	{attribute	'TcLinkTo'	:=	'.Status:=TIIB[LAMP_CLSTR1_PNL1_EP03_EP6002-0002]^COM TxPDO-Map Inputs Channel 1^Status;
								 .D[0]:=TIIB[LAMP_CLSTR1_PNL1_EP03_EP6002-0002]^COM TxPDO-Map Inputs Channel 1^Data In 0;
								 .D[1]:=TIIB[LAMP_CLSTR1_PNL1_EP03_EP6002-0002]^COM TxPDO-Map Inputs Channel 1^Data In 1;
								 .D[2]:=TIIB[LAMP_CLSTR1_PNL1_EP03_EP6002-0002]^COM TxPDO-Map Inputs Channel 1^Data In 2;
								 .D[3]:=TIIB[LAMP_CLSTR1_PNL1_EP03_EP6002-0002]^COM TxPDO-Map Inputs Channel 1^Data In 3;
								 .D[4]:=TIIB[LAMP_CLSTR1_PNL1_EP03_EP6002-0002]^COM TxPDO-Map Inputs Channel 1^Data In 4;
								 .D[5]:=TIIB[LAMP_CLSTR1_PNL1_EP03_EP6002-0002]^COM TxPDO-Map Inputs Channel 1^Data In 5;
								 .D[6]:=TIIB[LAMP_CLSTR1_PNL1_EP03_EP6002-0002]^COM TxPDO-Map Inputs Channel 1^Data In 6;
								 .D[7]:=TIIB[LAMP_CLSTR1_PNL1_EP03_EP6002-0002]^COM TxPDO-Map Inputs Channel 1^Data In 7;
								 .D[8]:=TIIB[LAMP_CLSTR1_PNL1_EP03_EP6002-0002]^COM TxPDO-Map Inputs Channel 1^Data In 8;
								 .D[9]:=TIIB[LAMP_CLSTR1_PNL1_EP03_EP6002-0002]^COM TxPDO-Map Inputs Channel 1^Data In 9;
								 .D[10]:=TIIB[LAMP_CLSTR1_PNL1_EP03_EP6002-0002]^COM TxPDO-Map Inputs Channel 1^Data In 10;
								 .D[11]:=TIIB[LAMP_CLSTR1_PNL1_EP03_EP6002-0002]^COM TxPDO-Map Inputs Channel 1^Data In 11;
								 .D[12]:=TIIB[LAMP_CLSTR1_PNL1_EP03_EP6002-0002]^COM TxPDO-Map Inputs Channel 1^Data In 12;
								 .D[13]:=TIIB[LAMP_CLSTR1_PNL1_EP03_EP6002-0002]^COM TxPDO-Map Inputs Channel 1^Data In 13;
								 .D[14]:=TIIB[LAMP_CLSTR1_PNL1_EP03_EP6002-0002]^COM TxPDO-Map Inputs Channel 1^Data In 14;
								 .D[15]:=TIIB[LAMP_CLSTR1_PNL1_EP03_EP6002-0002]^COM TxPDO-Map Inputs Channel 1^Data In 15;
								 .D[16]:=TIIB[LAMP_CLSTR1_PNL1_EP03_EP6002-0002]^COM TxPDO-Map Inputs Channel 1^Data In 16;
								 .D[17]:=TIIB[LAMP_CLSTR1_PNL1_EP03_EP6002-0002]^COM TxPDO-Map Inputs Channel 1^Data In 17;
								 .D[18]:=TIIB[LAMP_CLSTR1_PNL1_EP03_EP6002-0002]^COM TxPDO-Map Inputs Channel 1^Data In 18;
								 .D[19]:=TIIB[LAMP_CLSTR1_PNL1_EP03_EP6002-0002]^COM TxPDO-Map Inputs Channel 1^Data In 19;
								 .D[20]:=TIIB[LAMP_CLSTR1_PNL1_EP03_EP6002-0002]^COM TxPDO-Map Inputs Channel 1^Data In 20;
								 .D[21]:=TIIB[LAMP_CLSTR1_PNL1_EP03_EP6002-0002]^COM TxPDO-Map Inputs Channel 1^Data In 21
	'}
	stComIn_LAMP_CLSTR1_PTM_01		AT %I*	:	EL6inData22B;
	
	{attribute	'TcLinkTo'	:=	'.Ctrl:=TIIB[LAMP_CLSTR1_PNL1_EP03_EP6002-0002]^COM RxPDO-Map Outputs Channel 1^Ctrl;
								 .D[0]:=TIIB[LAMP_CLSTR1_PNL1_EP03_EP6002-0002]^COM RxPDO-Map Outputs Channel 1^Data Out 0;
								 .D[1]:=TIIB[LAMP_CLSTR1_PNL1_EP03_EP6002-0002]^COM RxPDO-Map Outputs Channel 1^Data Out 1;
								 .D[2]:=TIIB[LAMP_CLSTR1_PNL1_EP03_EP6002-0002]^COM RxPDO-Map Outputs Channel 1^Data Out 2;
								 .D[3]:=TIIB[LAMP_CLSTR1_PNL1_EP03_EP6002-0002]^COM RxPDO-Map Outputs Channel 1^Data Out 3;
								 .D[4]:=TIIB[LAMP_CLSTR1_PNL1_EP03_EP6002-0002]^COM RxPDO-Map Outputs Channel 1^Data Out 4;
								 .D[5]:=TIIB[LAMP_CLSTR1_PNL1_EP03_EP6002-0002]^COM RxPDO-Map Outputs Channel 1^Data Out 5;
								 .D[6]:=TIIB[LAMP_CLSTR1_PNL1_EP03_EP6002-0002]^COM RxPDO-Map Outputs Channel 1^Data Out 6;
								 .D[7]:=TIIB[LAMP_CLSTR1_PNL1_EP03_EP6002-0002]^COM RxPDO-Map Outputs Channel 1^Data Out 7;
								 .D[8]:=TIIB[LAMP_CLSTR1_PNL1_EP03_EP6002-0002]^COM RxPDO-Map Outputs Channel 1^Data Out 8;
								 .D[9]:=TIIB[LAMP_CLSTR1_PNL1_EP03_EP6002-0002]^COM RxPDO-Map Outputs Channel 1^Data Out 9;
								 .D[10]:=TIIB[LAMP_CLSTR1_PNL1_EP03_EP6002-0002]^COM RxPDO-Map Outputs Channel 1^Data Out 10;
								 .D[11]:=TIIB[LAMP_CLSTR1_PNL1_EP03_EP6002-0002]^COM RxPDO-Map Outputs Channel 1^Data Out 11;
								 .D[12]:=TIIB[LAMP_CLSTR1_PNL1_EP03_EP6002-0002]^COM RxPDO-Map Outputs Channel 1^Data Out 12;
								 .D[13]:=TIIB[LAMP_CLSTR1_PNL1_EP03_EP6002-0002]^COM RxPDO-Map Outputs Channel 1^Data Out 13;
								 .D[14]:=TIIB[LAMP_CLSTR1_PNL1_EP03_EP6002-0002]^COM RxPDO-Map Outputs Channel 1^Data Out 14;
								 .D[15]:=TIIB[LAMP_CLSTR1_PNL1_EP03_EP6002-0002]^COM RxPDO-Map Outputs Channel 1^Data Out 15;
								 .D[16]:=TIIB[LAMP_CLSTR1_PNL1_EP03_EP6002-0002]^COM RxPDO-Map Outputs Channel 1^Data Out 16;
								 .D[17]:=TIIB[LAMP_CLSTR1_PNL1_EP03_EP6002-0002]^COM RxPDO-Map Outputs Channel 1^Data Out 17;
								 .D[18]:=TIIB[LAMP_CLSTR1_PNL1_EP03_EP6002-0002]^COM RxPDO-Map Outputs Channel 1^Data Out 18;
								 .D[19]:=TIIB[LAMP_CLSTR1_PNL1_EP03_EP6002-0002]^COM RxPDO-Map Outputs Channel 1^Data Out 19;
								 .D[20]:=TIIB[LAMP_CLSTR1_PNL1_EP03_EP6002-0002]^COM RxPDO-Map Outputs Channel 1^Data Out 20;
								 .D[21]:=TIIB[LAMP_CLSTR1_PNL1_EP03_EP6002-0002]^COM RxPDO-Map Outputs Channel 1^Data Out 21
	'}
	stComOut_LAMP_CLSTR1_PTM_01		AT %Q*	:	EL6outData22B;
	
	{attribute	'TcLinkTo'	:=	'.Status:=TIIB[LAMP_CLSTR1_PNL2_EP03_EP6002-0002]^COM TxPDO-Map Inputs Channel 1^Status;
								 .D[0]:=TIIB[LAMP_CLSTR1_PNL2_EP03_EP6002-0002]^COM TxPDO-Map Inputs Channel 1^Data In 0;
								 .D[1]:=TIIB[LAMP_CLSTR1_PNL2_EP03_EP6002-0002]^COM TxPDO-Map Inputs Channel 1^Data In 1;
								 .D[2]:=TIIB[LAMP_CLSTR1_PNL2_EP03_EP6002-0002]^COM TxPDO-Map Inputs Channel 1^Data In 2;
								 .D[3]:=TIIB[LAMP_CLSTR1_PNL2_EP03_EP6002-0002]^COM TxPDO-Map Inputs Channel 1^Data In 3;
								 .D[4]:=TIIB[LAMP_CLSTR1_PNL2_EP03_EP6002-0002]^COM TxPDO-Map Inputs Channel 1^Data In 4;
								 .D[5]:=TIIB[LAMP_CLSTR1_PNL2_EP03_EP6002-0002]^COM TxPDO-Map Inputs Channel 1^Data In 5;
								 .D[6]:=TIIB[LAMP_CLSTR1_PNL2_EP03_EP6002-0002]^COM TxPDO-Map Inputs Channel 1^Data In 6;
								 .D[7]:=TIIB[LAMP_CLSTR1_PNL2_EP03_EP6002-0002]^COM TxPDO-Map Inputs Channel 1^Data In 7;
								 .D[8]:=TIIB[LAMP_CLSTR1_PNL2_EP03_EP6002-0002]^COM TxPDO-Map Inputs Channel 1^Data In 8;
								 .D[9]:=TIIB[LAMP_CLSTR1_PNL2_EP03_EP6002-0002]^COM TxPDO-Map Inputs Channel 1^Data In 9;
								 .D[10]:=TIIB[LAMP_CLSTR1_PNL2_EP03_EP6002-0002]^COM TxPDO-Map Inputs Channel 1^Data In 10;
								 .D[11]:=TIIB[LAMP_CLSTR1_PNL2_EP03_EP6002-0002]^COM TxPDO-Map Inputs Channel 1^Data In 11;
								 .D[12]:=TIIB[LAMP_CLSTR1_PNL2_EP03_EP6002-0002]^COM TxPDO-Map Inputs Channel 1^Data In 12;
								 .D[13]:=TIIB[LAMP_CLSTR1_PNL2_EP03_EP6002-0002]^COM TxPDO-Map Inputs Channel 1^Data In 13;
								 .D[14]:=TIIB[LAMP_CLSTR1_PNL2_EP03_EP6002-0002]^COM TxPDO-Map Inputs Channel 1^Data In 14;
								 .D[15]:=TIIB[LAMP_CLSTR1_PNL2_EP03_EP6002-0002]^COM TxPDO-Map Inputs Channel 1^Data In 15;
								 .D[16]:=TIIB[LAMP_CLSTR1_PNL2_EP03_EP6002-0002]^COM TxPDO-Map Inputs Channel 1^Data In 16;
								 .D[17]:=TIIB[LAMP_CLSTR1_PNL2_EP03_EP6002-0002]^COM TxPDO-Map Inputs Channel 1^Data In 17;
								 .D[18]:=TIIB[LAMP_CLSTR1_PNL2_EP03_EP6002-0002]^COM TxPDO-Map Inputs Channel 1^Data In 18;
								 .D[19]:=TIIB[LAMP_CLSTR1_PNL2_EP03_EP6002-0002]^COM TxPDO-Map Inputs Channel 1^Data In 19;
								 .D[20]:=TIIB[LAMP_CLSTR1_PNL2_EP03_EP6002-0002]^COM TxPDO-Map Inputs Channel 1^Data In 20;
								 .D[21]:=TIIB[LAMP_CLSTR1_PNL2_EP03_EP6002-0002]^COM TxPDO-Map Inputs Channel 1^Data In 21
	'}
	stComIn_LAMP_CLSTR1_PTM_02		AT %I*	:	EL6inData22B;
	
	{attribute	'TcLinkTo'	:=	'.Ctrl:=TIIB[LAMP_CLSTR1_PNL2_EP03_EP6002-0002]^COM RxPDO-Map Outputs Channel 1^Ctrl;
								 .D[0]:=TIIB[LAMP_CLSTR1_PNL2_EP03_EP6002-0002]^COM RxPDO-Map Outputs Channel 1^Data Out 0;
								 .D[1]:=TIIB[LAMP_CLSTR1_PNL2_EP03_EP6002-0002]^COM RxPDO-Map Outputs Channel 1^Data Out 1;
								 .D[2]:=TIIB[LAMP_CLSTR1_PNL2_EP03_EP6002-0002]^COM RxPDO-Map Outputs Channel 1^Data Out 2;
								 .D[3]:=TIIB[LAMP_CLSTR1_PNL2_EP03_EP6002-0002]^COM RxPDO-Map Outputs Channel 1^Data Out 3;
								 .D[4]:=TIIB[LAMP_CLSTR1_PNL2_EP03_EP6002-0002]^COM RxPDO-Map Outputs Channel 1^Data Out 4;
								 .D[5]:=TIIB[LAMP_CLSTR1_PNL2_EP03_EP6002-0002]^COM RxPDO-Map Outputs Channel 1^Data Out 5;
								 .D[6]:=TIIB[LAMP_CLSTR1_PNL2_EP03_EP6002-0002]^COM RxPDO-Map Outputs Channel 1^Data Out 6;
								 .D[7]:=TIIB[LAMP_CLSTR1_PNL2_EP03_EP6002-0002]^COM RxPDO-Map Outputs Channel 1^Data Out 7;
								 .D[8]:=TIIB[LAMP_CLSTR1_PNL2_EP03_EP6002-0002]^COM RxPDO-Map Outputs Channel 1^Data Out 8;
								 .D[9]:=TIIB[LAMP_CLSTR1_PNL2_EP03_EP6002-0002]^COM RxPDO-Map Outputs Channel 1^Data Out 9;
								 .D[10]:=TIIB[LAMP_CLSTR1_PNL2_EP03_EP6002-0002]^COM RxPDO-Map Outputs Channel 1^Data Out 10;
								 .D[11]:=TIIB[LAMP_CLSTR1_PNL2_EP03_EP6002-0002]^COM RxPDO-Map Outputs Channel 1^Data Out 11;
								 .D[12]:=TIIB[LAMP_CLSTR1_PNL2_EP03_EP6002-0002]^COM RxPDO-Map Outputs Channel 1^Data Out 12;
								 .D[13]:=TIIB[LAMP_CLSTR1_PNL2_EP03_EP6002-0002]^COM RxPDO-Map Outputs Channel 1^Data Out 13;
								 .D[14]:=TIIB[LAMP_CLSTR1_PNL2_EP03_EP6002-0002]^COM RxPDO-Map Outputs Channel 1^Data Out 14;
								 .D[15]:=TIIB[LAMP_CLSTR1_PNL2_EP03_EP6002-0002]^COM RxPDO-Map Outputs Channel 1^Data Out 15;
								 .D[16]:=TIIB[LAMP_CLSTR1_PNL2_EP03_EP6002-0002]^COM RxPDO-Map Outputs Channel 1^Data Out 16;
								 .D[17]:=TIIB[LAMP_CLSTR1_PNL2_EP03_EP6002-0002]^COM RxPDO-Map Outputs Channel 1^Data Out 17;
								 .D[18]:=TIIB[LAMP_CLSTR1_PNL2_EP03_EP6002-0002]^COM RxPDO-Map Outputs Channel 1^Data Out 18;
								 .D[19]:=TIIB[LAMP_CLSTR1_PNL2_EP03_EP6002-0002]^COM RxPDO-Map Outputs Channel 1^Data Out 19;
								 .D[20]:=TIIB[LAMP_CLSTR1_PNL2_EP03_EP6002-0002]^COM RxPDO-Map Outputs Channel 1^Data Out 20;
								 .D[21]:=TIIB[LAMP_CLSTR1_PNL2_EP03_EP6002-0002]^COM RxPDO-Map Outputs Channel 1^Data Out 21
	'}
	stComOut_LAMP_CLSTR1_PTM_02		AT %Q*	:	EL6outData22B;
	
	{attribute	'TcLinkTo'	:=	'.Status:=TIIB[LAMP_CLSTR1_PNL3_EP03_EP6002-0002]^COM TxPDO-Map Inputs Channel 1^Status;
								 .D[0]:=TIIB[LAMP_CLSTR1_PNL3_EP03_EP6002-0002]^COM TxPDO-Map Inputs Channel 1^Data In 0;
								 .D[1]:=TIIB[LAMP_CLSTR1_PNL3_EP03_EP6002-0002]^COM TxPDO-Map Inputs Channel 1^Data In 1;
								 .D[2]:=TIIB[LAMP_CLSTR1_PNL3_EP03_EP6002-0002]^COM TxPDO-Map Inputs Channel 1^Data In 2;
								 .D[3]:=TIIB[LAMP_CLSTR1_PNL3_EP03_EP6002-0002]^COM TxPDO-Map Inputs Channel 1^Data In 3;
								 .D[4]:=TIIB[LAMP_CLSTR1_PNL3_EP03_EP6002-0002]^COM TxPDO-Map Inputs Channel 1^Data In 4;
								 .D[5]:=TIIB[LAMP_CLSTR1_PNL3_EP03_EP6002-0002]^COM TxPDO-Map Inputs Channel 1^Data In 5;
								 .D[6]:=TIIB[LAMP_CLSTR1_PNL3_EP03_EP6002-0002]^COM TxPDO-Map Inputs Channel 1^Data In 6;
								 .D[7]:=TIIB[LAMP_CLSTR1_PNL3_EP03_EP6002-0002]^COM TxPDO-Map Inputs Channel 1^Data In 7;
								 .D[8]:=TIIB[LAMP_CLSTR1_PNL3_EP03_EP6002-0002]^COM TxPDO-Map Inputs Channel 1^Data In 8;
								 .D[9]:=TIIB[LAMP_CLSTR1_PNL3_EP03_EP6002-0002]^COM TxPDO-Map Inputs Channel 1^Data In 9;
								 .D[10]:=TIIB[LAMP_CLSTR1_PNL3_EP03_EP6002-0002]^COM TxPDO-Map Inputs Channel 1^Data In 10;
								 .D[11]:=TIIB[LAMP_CLSTR1_PNL3_EP03_EP6002-0002]^COM TxPDO-Map Inputs Channel 1^Data In 11;
								 .D[12]:=TIIB[LAMP_CLSTR1_PNL3_EP03_EP6002-0002]^COM TxPDO-Map Inputs Channel 1^Data In 12;
								 .D[13]:=TIIB[LAMP_CLSTR1_PNL3_EP03_EP6002-0002]^COM TxPDO-Map Inputs Channel 1^Data In 13;
								 .D[14]:=TIIB[LAMP_CLSTR1_PNL3_EP03_EP6002-0002]^COM TxPDO-Map Inputs Channel 1^Data In 14;
								 .D[15]:=TIIB[LAMP_CLSTR1_PNL3_EP03_EP6002-0002]^COM TxPDO-Map Inputs Channel 1^Data In 15;
								 .D[16]:=TIIB[LAMP_CLSTR1_PNL3_EP03_EP6002-0002]^COM TxPDO-Map Inputs Channel 1^Data In 16;
								 .D[17]:=TIIB[LAMP_CLSTR1_PNL3_EP03_EP6002-0002]^COM TxPDO-Map Inputs Channel 1^Data In 17;
								 .D[18]:=TIIB[LAMP_CLSTR1_PNL3_EP03_EP6002-0002]^COM TxPDO-Map Inputs Channel 1^Data In 18;
								 .D[19]:=TIIB[LAMP_CLSTR1_PNL3_EP03_EP6002-0002]^COM TxPDO-Map Inputs Channel 1^Data In 19;
								 .D[20]:=TIIB[LAMP_CLSTR1_PNL3_EP03_EP6002-0002]^COM TxPDO-Map Inputs Channel 1^Data In 20;
								 .D[21]:=TIIB[LAMP_CLSTR1_PNL3_EP03_EP6002-0002]^COM TxPDO-Map Inputs Channel 1^Data In 21
	'}
	stComIn_LAMP_CLSTR1_PTM_03		AT %I*	:	EL6inData22B;
	
	{attribute	'TcLinkTo'	:=	'.Ctrl:=TIIB[LAMP_CLSTR1_PNL3_EP03_EP6002-0002]^COM RxPDO-Map Outputs Channel 1^Ctrl;
								 .D[0]:=TIIB[LAMP_CLSTR1_PNL3_EP03_EP6002-0002]^COM RxPDO-Map Outputs Channel 1^Data Out 0;
								 .D[1]:=TIIB[LAMP_CLSTR1_PNL3_EP03_EP6002-0002]^COM RxPDO-Map Outputs Channel 1^Data Out 1;
								 .D[2]:=TIIB[LAMP_CLSTR1_PNL3_EP03_EP6002-0002]^COM RxPDO-Map Outputs Channel 1^Data Out 2;
								 .D[3]:=TIIB[LAMP_CLSTR1_PNL3_EP03_EP6002-0002]^COM RxPDO-Map Outputs Channel 1^Data Out 3;
								 .D[4]:=TIIB[LAMP_CLSTR1_PNL3_EP03_EP6002-0002]^COM RxPDO-Map Outputs Channel 1^Data Out 4;
								 .D[5]:=TIIB[LAMP_CLSTR1_PNL3_EP03_EP6002-0002]^COM RxPDO-Map Outputs Channel 1^Data Out 5;
								 .D[6]:=TIIB[LAMP_CLSTR1_PNL3_EP03_EP6002-0002]^COM RxPDO-Map Outputs Channel 1^Data Out 6;
								 .D[7]:=TIIB[LAMP_CLSTR1_PNL3_EP03_EP6002-0002]^COM RxPDO-Map Outputs Channel 1^Data Out 7;
								 .D[8]:=TIIB[LAMP_CLSTR1_PNL3_EP03_EP6002-0002]^COM RxPDO-Map Outputs Channel 1^Data Out 8;
								 .D[9]:=TIIB[LAMP_CLSTR1_PNL3_EP03_EP6002-0002]^COM RxPDO-Map Outputs Channel 1^Data Out 9;
								 .D[10]:=TIIB[LAMP_CLSTR1_PNL3_EP03_EP6002-0002]^COM RxPDO-Map Outputs Channel 1^Data Out 10;
								 .D[11]:=TIIB[LAMP_CLSTR1_PNL3_EP03_EP6002-0002]^COM RxPDO-Map Outputs Channel 1^Data Out 11;
								 .D[12]:=TIIB[LAMP_CLSTR1_PNL3_EP03_EP6002-0002]^COM RxPDO-Map Outputs Channel 1^Data Out 12;
								 .D[13]:=TIIB[LAMP_CLSTR1_PNL3_EP03_EP6002-0002]^COM RxPDO-Map Outputs Channel 1^Data Out 13;
								 .D[14]:=TIIB[LAMP_CLSTR1_PNL3_EP03_EP6002-0002]^COM RxPDO-Map Outputs Channel 1^Data Out 14;
								 .D[15]:=TIIB[LAMP_CLSTR1_PNL3_EP03_EP6002-0002]^COM RxPDO-Map Outputs Channel 1^Data Out 15;
								 .D[16]:=TIIB[LAMP_CLSTR1_PNL3_EP03_EP6002-0002]^COM RxPDO-Map Outputs Channel 1^Data Out 16;
								 .D[17]:=TIIB[LAMP_CLSTR1_PNL3_EP03_EP6002-0002]^COM RxPDO-Map Outputs Channel 1^Data Out 17;
								 .D[18]:=TIIB[LAMP_CLSTR1_PNL3_EP03_EP6002-0002]^COM RxPDO-Map Outputs Channel 1^Data Out 18;
								 .D[19]:=TIIB[LAMP_CLSTR1_PNL3_EP03_EP6002-0002]^COM RxPDO-Map Outputs Channel 1^Data Out 19;
								 .D[20]:=TIIB[LAMP_CLSTR1_PNL3_EP03_EP6002-0002]^COM RxPDO-Map Outputs Channel 1^Data Out 20;
								 .D[21]:=TIIB[LAMP_CLSTR1_PNL3_EP03_EP6002-0002]^COM RxPDO-Map Outputs Channel 1^Data Out 21
	'}
	stComOut_LAMP_CLSTR1_PTM_03		AT %Q*	:	EL6outData22B;
(*
	{attribute	'TcLinkTo'	:=	'.Status:=TIIB[KTOF_PNL1_EP03_EP6002-0002]^COM TxPDO-Map Inputs Channel 1^Status;
								 .D[0]:=TIIB[KTOF_PNL1_EP03_EP6002-0002]^COM TxPDO-Map Inputs Channel 1^Data In 0;
								 .D[1]:=TIIB[KTOF_PNL1_EP03_EP6002-0002]^COM TxPDO-Map Inputs Channel 1^Data In 1;
								 .D[2]:=TIIB[KTOF_PNL1_EP03_EP6002-0002]^COM TxPDO-Map Inputs Channel 1^Data In 2;
								 .D[3]:=TIIB[KTOF_PNL1_EP03_EP6002-0002]^COM TxPDO-Map Inputs Channel 1^Data In 3;
								 .D[4]:=TIIB[KTOF_PNL1_EP03_EP6002-0002]^COM TxPDO-Map Inputs Channel 1^Data In 4;
								 .D[5]:=TIIB[KTOF_PNL1_EP03_EP6002-0002]^COM TxPDO-Map Inputs Channel 1^Data In 5;
								 .D[6]:=TIIB[KTOF_PNL1_EP03_EP6002-0002]^COM TxPDO-Map Inputs Channel 1^Data In 6;
								 .D[7]:=TIIB[KTOF_PNL1_EP03_EP6002-0002]^COM TxPDO-Map Inputs Channel 1^Data In 7;
								 .D[8]:=TIIB[KTOF_PNL1_EP03_EP6002-0002]^COM TxPDO-Map Inputs Channel 1^Data In 8;
								 .D[9]:=TIIB[KTOF_PNL1_EP03_EP6002-0002]^COM TxPDO-Map Inputs Channel 1^Data In 9;
								 .D[10]:=TIIB[KTOF_PNL1_EP03_EP6002-0002]^COM TxPDO-Map Inputs Channel 1^Data In 10;
								 .D[11]:=TIIB[KTOF_PNL1_EP03_EP6002-0002]^COM TxPDO-Map Inputs Channel 1^Data In 11;
								 .D[12]:=TIIB[KTOF_PNL1_EP03_EP6002-0002]^COM TxPDO-Map Inputs Channel 1^Data In 12;
								 .D[13]:=TIIB[KTOF_PNL1_EP03_EP6002-0002]^COM TxPDO-Map Inputs Channel 1^Data In 13;
								 .D[14]:=TIIB[KTOF_PNL1_EP03_EP6002-0002]^COM TxPDO-Map Inputs Channel 1^Data In 14;
								 .D[15]:=TIIB[KTOF_PNL1_EP03_EP6002-0002]^COM TxPDO-Map Inputs Channel 1^Data In 15;
								 .D[16]:=TIIB[KTOF_PNL1_EP03_EP6002-0002]^COM TxPDO-Map Inputs Channel 1^Data In 16;
								 .D[17]:=TIIB[KTOF_PNL1_EP03_EP6002-0002]^COM TxPDO-Map Inputs Channel 1^Data In 17;
								 .D[18]:=TIIB[KTOF_PNL1_EP03_EP6002-0002]^COM TxPDO-Map Inputs Channel 1^Data In 18;
								 .D[19]:=TIIB[KTOF_PNL1_EP03_EP6002-0002]^COM TxPDO-Map Inputs Channel 1^Data In 19;
								 .D[20]:=TIIB[KTOF_PNL1_EP03_EP6002-0002]^COM TxPDO-Map Inputs Channel 1^Data In 20;
								 .D[21]:=TIIB[KTOF_PNL1_EP03_EP6002-0002]^COM TxPDO-Map Inputs Channel 1^Data In 21;
	'}
	stComIn_KTOF_PTM_01		AT %I*	:	EL6inData22B;

	{attribute	'TcLinkTo'	:=	'.Ctrl:=TIIB[KTOF_PNL1_EP03_EP6002-0002]^COM RxPDO-Map Outputs Channel 1^Ctrl;
								 .D[0]:=TIIB[KTOF_PNL1_EP03_EP6002-0002]^COM RxPDO-Map Outputs Channel 1^Data Out 0;
								 .D[1]:=TIIB[KTOF_PNL1_EP03_EP6002-0002]^COM RxPDO-Map Outputs Channel 1^Data Out 1;
								 .D[2]:=TIIB[KTOF_PNL1_EP03_EP6002-0002]^COM RxPDO-Map Outputs Channel 1^Data Out 2;
								 .D[3]:=TIIB[KTOF_PNL1_EP03_EP6002-0002]^COM RxPDO-Map Outputs Channel 1^Data Out 3;
								 .D[4]:=TIIB[KTOF_PNL1_EP03_EP6002-0002]^COM RxPDO-Map Outputs Channel 1^Data Out 4;
								 .D[5]:=TIIB[KTOF_PNL1_EP03_EP6002-0002]^COM RxPDO-Map Outputs Channel 1^Data Out 5;
								 .D[6]:=TIIB[KTOF_PNL1_EP03_EP6002-0002]^COM RxPDO-Map Outputs Channel 1^Data Out 6;
								 .D[7]:=TIIB[KTOF_PNL1_EP03_EP6002-0002]^COM RxPDO-Map Outputs Channel 1^Data Out 7;
								 .D[8]:=TIIB[KTOF_PNL1_EP03_EP6002-0002]^COM RxPDO-Map Outputs Channel 1^Data Out 8;
								 .D[9]:=TIIB[KTOF_PNL1_EP03_EP6002-0002]^COM RxPDO-Map Outputs Channel 1^Data Out 9;
								 .D[10]:=TIIB[KTOF_PNL1_EP03_EP6002-0002]^COM RxPDO-Map Outputs Channel 1^Data Out 10;
								 .D[11]:=TIIB[KTOF_PNL1_EP03_EP6002-0002]^COM RxPDO-Map Outputs Channel 1^Data Out 11;
								 .D[12]:=TIIB[KTOF_PNL1_EP03_EP6002-0002]^COM RxPDO-Map Outputs Channel 1^Data Out 12;
								 .D[13]:=TIIB[KTOF_PNL1_EP03_EP6002-0002]^COM RxPDO-Map Outputs Channel 1^Data Out 13;
								 .D[14]:=TIIB[KTOF_PNL1_EP03_EP6002-0002]^COM RxPDO-Map Outputs Channel 1^Data Out 14;
								 .D[15]:=TIIB[KTOF_PNL1_EP03_EP6002-0002]^COM RxPDO-Map Outputs Channel 1^Data Out 15;
								 .D[16]:=TIIB[KTOF_PNL1_EP03_EP6002-0002]^COM RxPDO-Map Outputs Channel 1^Data Out 16;
								 .D[17]:=TIIB[KTOF_PNL1_EP03_EP6002-0002]^COM RxPDO-Map Outputs Channel 1^Data Out 17;
								 .D[18]:=TIIB[KTOF_PNL1_EP03_EP6002-0002]^COM RxPDO-Map Outputs Channel 1^Data Out 18;
								 .D[19]:=TIIB[KTOF_PNL1_EP03_EP6002-0002]^COM RxPDO-Map Outputs Channel 1^Data Out 19;
								 .D[20]:=TIIB[KTOF_PNL1_EP03_EP6002-0002]^COM RxPDO-Map Outputs Channel 1^Data Out 20;
								 .D[21]:=TIIB[KTOF_PNL1_EP03_EP6002-0002]^COM RxPDO-Map Outputs Channel 1^Data Out 21;
	'}
	stComOut_KTOF_PTM_01		AT %Q*	:	EL6outData22B;
*)
	//Leybolds
	// GJ2 not included in LV17 configuration
END_VAR

// ---- GVLs/GVL_Devices.TcGVL
//{attribute 'qualified_only'}
VAR_GLOBAL
	
(*Rack Mounted Turbo Pumps*)
// GJ2 not included in LV17 configuration

(*Onboard Turbo Pumps*)
	{attribute 'TcLinkTo' := 	'.i_xAtSpd			:=	TIIB[LAMP_PNL1_EP01_EP2338-0002]^Channel 1^Input;
								 .i_xFaultNC		:=	TIIB[LAMP_PNL1_EP01_EP2338-0002]^Channel 2^Input;
								 .i_xRemote			:=	TIIB[LAMP_PNL1_EP01_EP2338-0002]^Channel 3^Input;
								 .q_RunDO			:=	TIIB[LAMP_PNL1_EP02_EP2624-0002]^Channel 1^Output;
								 .q_xReset 			:=	TIIB[LAMP_PNL1_EP02_EP2624-0002]^Channel 2^Output				 
	'}
	{attribute 'pytmc' := '
		pv: LAMP:C2:PTM:01
		io: io
	'}
	LAMP_C2_PTM_01 : FB_PTM_Pfeiffer;
	
	{attribute 'TcLinkTo' := 	'.i_xAtSpd			:=	TIIB[LAMP_PNL1_EP01_EP2338-0002]^Channel 5^Input;
								 .i_xFaultNC		:=	TIIB[LAMP_PNL1_EP01_EP2338-0002]^Channel 6^Input;
								 .i_xRemote			:=	TIIB[LAMP_PNL1_EP01_EP2338-0002]^Channel 7^Input;
								 .q_RunDO			:=	TIIB[LAMP_PNL1_EP02_EP2624-0002]^Channel 3^Output;
								 .q_xReset 			:=	TIIB[LAMP_PNL1_EP02_EP2624-0002]^Channel 4^Output				 
	'}
	{attribute 'pytmc' := '
		pv: LAMP:C2:PTM:02
		io: io
	'}
	LAMP_C2_PTM_02 : FB_PTM_Pfeiffer;
	
	{attribute 'TcLinkTo' := 	'.i_xAtSpd			:=	TIIB[LAMP_PNL1_EP04_EP2338-0002]^Channel 1^Input;
								 .i_xFaultNC		:=	TIIB[LAMP_PNL1_EP04_EP2338-0002]^Channel 2^Input;
								 .i_xRemote			:=	TIIB[LAMP_PNL1_EP04_EP2338-0002]^Channel 3^Input;
								 .q_RunDO			:=	TIIB[LAMP_PNL1_EP05_EP2624-0002]^Channel 1^Output;
								 .q_xReset 			:=	TIIB[LAMP_PNL1_EP05_EP2624-0002]^Channel 2^Output				 
	'}
	{attribute 'pytmc' := '
		pv: LAMP:C2:PTM:03
		io: io
	'}
	LAMP_C2_PTM_03 : FB_PTM_Pfeiffer;
	
	{attribute 'TcLinkTo' := 	'.i_xAtSpd			:=	TIIB[LAMP_PNL1_EP04_EP2338-0002]^Channel 5^Input;
								 .i_xFaultNC		:=	TIIB[LAMP_PNL1_EP04_EP2338-0002]^Channel 6^Input;
								 .i_xRemote			:=	TIIB[LAMP_PNL1_EP04_EP2338-0002]^Channel 7^Input;
								 .q_RunDO			:=	TIIB[LAMP_PNL1_EP05_EP2624-0002]^Channel 3^Output;
								 .q_xReset 			:=	TIIB[LAMP_PNL1_EP05_EP2624-0002]^Channel 4^Output				 
	'}
	{attribute 'pytmc' := '
		pv: LAMP:C2:PTM:04
		io: io
	'}
	LAMP_C2_PTM_04 : FB_PTM_Pfeiffer;
	
	{attribute 'TcLinkTo' := 	'.i_xAtSpd			:=	TIIB[LAMP_PNL2_EP16_EP2338-0002]^Channel 1^Input;
								 .i_xFaultNC		:=	TIIB[LAMP_PNL2_EP16_EP2338-0002]^Channel 2^Input;
								 .q_RunDO			:=	TIIB[LAMP_PNL2_EP17_EP2624-0002]^Channel 1^Output;
								 .q_xReset 			:=	TIIB[LAMP_PNL2_EP17_EP2624-0002]^Channel 2^Output				 
	'}
	{attribute 'pytmc' := '
		pv: LAMP:CATCH:PTM:01
		io: io
	'}
	LAMP_CATCH_PTM_01 : FB_PTM_Pfeiffer;
	
	{attribute 'TcLinkTo' := 	'.i_xAtSpd			:=	TIIB[LAMP_PNL2_EP16_EP2338-0002]^Channel 5^Input;
								 .i_xFaultNC		:=	TIIB[LAMP_PNL2_EP16_EP2338-0002]^Channel 6^Input;
								 .q_RunDO			:=	TIIB[LAMP_PNL2_EP17_EP2624-0002]^Channel 3^Output;
								 .q_xReset 			:=	TIIB[LAMP_PNL2_EP17_EP2624-0002]^Channel 4^Output				 
	'}
	{attribute 'pytmc' := '
		pv: LAMP:CATCH:PTM:02
		io: io
	'}
	LAMP_CATCH_PTM_02 : FB_PTM_Pfeiffer;
	
	{attribute 'TcLinkTo' := 	'.i_xAtSpd			:=	TIIB[LAMP_PNL2_EP13_EP2338-0002]^Channel 1^Input;
								 .i_xFaultNC		:=	TIIB[LAMP_PNL2_EP13_EP2338-0002]^Channel 2^Input;
								 .i_xRemote			:=	TIIB[LAMP_PNL2_EP13_EP2338-0002]^Channel 3^Input;
								 .q_RunDO			:=	TIIB[LAMP_PNL2_EP14_EP2624-0002]^Channel 1^Output;
								 .q_xReset 			:=	TIIB[LAMP_PNL2_EP14_EP2624-0002]^Channel 2^Output				 
	'}
	{attribute 'pytmc' := '
		pv: LAMP:ROUGH:PTM:01
		io: io
	'}
	LAMP_ROUGH_PTM_01 : FB_PTM_Pfeiffer;
	
	{attribute 'TcLinkTo' := 	'.i_xAtSpd			:=	TIIB[LAMP_PNL2_EP13_EP2338-0002]^Channel 5^Input;
								 .i_xFaultNC		:=	TIIB[LAMP_PNL2_EP13_EP2338-0002]^Channel 6^Input;
								 .i_xRemote			:=	TIIB[LAMP_PNL2_EP13_EP2338-0002]^Channel 7^Input;
								 .q_RunDO			:=	TIIB[LAMP_PNL2_EP14_EP2624-0002]^Channel 3^Output;
								 .q_xReset 			:=	TIIB[LAMP_PNL2_EP14_EP2624-0002]^Channel 4^Output				 
	'}
	{attribute 'pytmc' := '
		pv: LAMP:C1:PTM:01
		io: io
	'}
	LAMP_C1_PTM_01 : FB_PTM_Pfeiffer;
	
// Cluster Source Turbo Pumps, LV17 Configuration

	{attribute 'TcLinkTo' := 	'.i_xAtSpd			:=	TIIB[LAMP_CLSTR1_PNL1_EP01_EP2338-0002]^Channel 1^Input;
								 .i_xFaultNC		:=	TIIB[LAMP_CLSTR1_PNL1_EP01_EP2338-0002]^Channel 2^Input;
								 .i_xRemote			:=	TIIB[LAMP_CLSTR1_PNL1_EP01_EP2338-0002]^Channel 3^Input;
								 .q_RunDO			:=	TIIB[LAMP_CLSTR1_PNL1_EP02_EP2624-0002]^Channel 1^Output;
								 .q_xReset 			:=	TIIB[LAMP_CLSTR1_PNL1_EP02_EP2624-0002]^Channel 2^Output				 
	'}
	{attribute 'pytmc' := '
		pv: LAMP:CLSTR1:PTM:01
		io: io
	'}
	LAMP_CLSTR1_PTM_01 : FB_PTM_Pfeiffer;	

	{attribute 'TcLinkTo' := 	'.i_xAtSpd			:=	TIIB[LAMP_CLSTR1_PNL2_EP01_EP2338-0002]^Channel 1^Input;
								 .i_xFaultNC		:=	TIIB[LAMP_CLSTR1_PNL2_EP01_EP2338-0002]^Channel 2^Input;
								 .i_xRemote			:=	TIIB[LAMP_CLSTR1_PNL2_EP01_EP2338-0002]^Channel 3^Input;
								 .q_RunDO			:=	TIIB[LAMP_CLSTR1_PNL2_EP02_EP2624-0002]^Channel 1^Output;
								 .q_xReset 			:=	TIIB[LAMP_CLSTR1_PNL2_EP02_EP2624-0002]^Channel 2^Output				 
	'}
	{attribute 'pytmc' := '
		pv: LAMP:CLSTR1:PTM:02
		io: io
	'}
	LAMP_CLSTR1_PTM_02 : FB_PTM_Pfeiffer;
	
	{attribute 'TcLinkTo' := 	'.i_xAtSpd			:=	TIIB[LAMP_CLSTR1_PNL3_EP01_EP2338-0002]^Channel 1^Input;
								 .i_xFaultNC		:=	TIIB[LAMP_CLSTR1_PNL3_EP01_EP2338-0002]^Channel 2^Input;
								 .i_xRemote			:=	TIIB[LAMP_CLSTR1_PNL3_EP01_EP2338-0002]^Channel 3^Input;
								 .q_RunDO			:=	TIIB[LAMP_CLSTR1_PNL3_EP02_EP2624-0002]^Channel 1^Output;
								 .q_xReset 			:=	TIIB[LAMP_CLSTR1_PNL3_EP02_EP2624-0002]^Channel 2^Output				 
	'}
	{attribute 'pytmc' := '
		pv: LAMP:CLSTR1:PTM:03
		io: io
	'}
	LAMP_CLSTR1_PTM_03 : FB_PTM_Pfeiffer;
	
(*KTOF Turbo Pump*)
(*
	{attribute 'TcLinkTo' := 	'.i_xAtSpd			:=	TIIB[KTOF_PNL1_EP01_EP2338-0002]^Channel 1^Input;
								 .i_xFaultNC		:=	TIIB[KTOF_PNL1_EP01_EP2338-0002]^Channel 2^Input;
								 .i_xRemote			:=	TIIB[KTOF_PNL1_EP01_EP2338-0002]^Channel 3^Input;
								 .q_RunDO			:=	TIIB[KTOF_PNL1_EP02_EP2624-0002]^Channel 1^Output;
								 .q_xReset 			:=	TIIB[KTOF_PNL1_EP02_EP2624-0002]^Channel 2^Output				 
	'}
	{attribute 'pytmc' := '
		pv: KTOF:PTM:01
		io: io
	'}
	KTOF_PTM_01 : FB_PTM_Pfeiffer;
*)
(*Pirani MKS 275 Gauges*)
	{attribute 'TcLinkTo' := 	'.i_iPRESS_R	:=	TIIB[LAMP_PNL2_EP19_EP3174-0002]^AI Standard Channel 1^Value
	'}
	{attribute 'pytmc' := '
		pv: LAMP:C2:GPI:01
		io: io
	'}
	LAMP_C2_GPI_01 : FB_MKS275;
	
(*	{attribute 'TcLinkTo' := 	'.i_iPRESS_R	:=	TIIB[LAMP_PNL2_EP19_EP3174-0002]^AI Standard Channel 2^Value
	'}
	{attribute 'pytmc' := '
		pv: LAMP:CATCH:GPI:01
		io: io
	'}
	LAMP_CATCH_GPI_01 : FB_MKS275; //NO GAUGE INSTALLED
*)	
	
	{attribute 'TcLinkTo' := 	'.i_iPRESS_R	:=	TIIB[LAMP_PNL2_EP19_EP3174-0002]^AI Standard Channel 3^Value
	'}
	{attribute 'pytmc' := '
		pv: LAMP:GJ1:GPI:01
		io: io
	'}
	LAMP_GJ1_GPI_01 : FB_MKS275;
	
	{attribute 'TcLinkTo' := 	'.i_iPRESS_R	:=	TIIB[LAMP_PNL2_EP19_EP3174-0002]^AI Standard Channel 4^Value
	'}
	{attribute 'pytmc' := '
		pv: LAMP:GJ2:GPI:01
		io: io
	'}
	LAMP_GJ2_GPI_01 : FB_MKS275;

(*MicroPirani MKS 925 Gauges*)
	{attribute 'TcLinkTo' := 	'.i_iPRESS_R	:=	TIIB[LAMP_PNL2_EP20_EP3174-0002]^AI Standard Channel 1^Value
	'}
	{attribute 'pytmc' := '
		pv: LAMP:ROUGH:GPI:01
		io: io
	'}
	LAMP_ROUGH_GPI_01 : FB_9XX;
	
	{attribute 'TcLinkTo' := 	'.i_iPRESS_R	:=	TIIB[LAMP_PNL2_EP20_EP3174-0002]^AI Standard Channel 2^Value
	'}
	{attribute 'pytmc' := '
		pv: LAMP:ROUGH:GPI:02
		io: io
	'}
	LAMP_ROUGH_GPI_02 : FB_9XX;
	
	{attribute 'TcLinkTo' := 	'.i_iPRESS_R	:=	TIIB[LAMP_PNL2_EP20_EP3174-0002]^AI Standard Channel 3^Value
	'}
	{attribute 'pytmc' := '
		pv: LAMP:ROUGH:GPI:03
		io: io
	'}
	LAMP_ROUGH_GPI_03 : FB_9XX;
	
	{attribute 'TcLinkTo' := 	'.i_iPRESS_R	:=	TIIB[LAMP_PNL2_EP20_EP3174-0002]^AI Standard Channel 4^Value
	'}
	{attribute 'pytmc' := '
		pv: LAMP:ROUGH:GPI:04
		io: io
	'}
	LAMP_ROUGH_GPI_04 : FB_9XX;

(*Cold Cathode MKS 500 Gauges*)
	{attribute 'TcLinkTo' := 	'.i_iPRESS_R	:=	TIIB[LAMP_PNL2_EP21_EP3174-0002]^AI Standard Channel 1^Value;
								 .q_xHV_DIS		:= 	TIIB[LAMP_PNL2_EP22_EP2624-0002]^Channel 1^Output
	'}	
	{attribute 'pytmc' := '
		pv: LAMP:C2:GCC:01
		io: io
	'}
	LAMP_C2_GCC_01 : FB_MKS500;
	
	{attribute 'TcLinkTo' := 	'.i_iPRESS_R	:=	TIIB[LAMP_PNL2_EP21_EP3174-0002]^AI Standard Channel 2^Value;
								 .q_xHV_DIS		:= 	TIIB[LAMP_PNL2_EP22_EP2624-0002]^Channel 2^Output
	'}	
	{attribute 'pytmc' := '
		pv: LAMP:CATCH:GCC:01
		io: io
	'}
	LAMP_CATCH_GCC_01 : FB_MKS500;
	
	{attribute 'TcLinkTo' := 	'.i_iPRESS_R	:=	TIIB[LAMP_PNL2_EP21_EP3174-0002]^AI Standard Channel 3^Value;
								 .q_xHV_DIS		:= 	TIIB[LAMP_PNL2_EP22_EP2624-0002]^Channel 3^Output
	'}	
	{attribute 'pytmc' := '
		pv: LAMP:CATCH:GCC:02
		io: io
	'}
	LAMP_CATCH_GCC_02 : FB_MKS500;
	
	{attribute 'TcLinkTo' := 	'.i_iPRESS_R	:=	TIIB[LAMP_PNL2_EP21_EP3174-0002]^AI Standard Channel 4^Value;
								 .q_xHV_DIS		:= 	TIIB[LAMP_PNL2_EP22_EP2624-0002]^Channel 4^Output
	'}	
	{attribute 'pytmc' := '
		pv: LAMP:GJ1:GCC:01
		io: io
	'}
	LAMP_GJ1_GCC_01 : FB_MKS500;
	
	{attribute 'TcLinkTo' := 	'.i_iPRESS_R	:=	TIIB[LAMP_PNL2_EP23_EP3174-0002]^AI Standard Channel 1^Value;
								 .q_xHV_DIS		:= 	TIIB[LAMP_PNL2_EP24_EP2624-0002]^Channel 1^Output
	'}	
	{attribute 'pytmc' := '
		pv: LAMP:GJ2:GCC:01
		io: io
	'}
	LAMP_GJ2_GCC_01 : FB_MKS500;

(*Hot Cathode MKS 909 Gauges*)
	{attribute 'TcLinkTo' := 	'.i_iPRESS_R	:=	TIIB[LAMP_PNL2_EP23_EP3174-0002]^AI Standard Channel 2^Value;
								 .q_xHV_DIS		:= 	TIIB[LAMP_PNL2_EP24_EP2624-0002]^Channel 2^Output
	'}	
	{attribute 'pytmc' := '
		pv: LAMP:C1:GHC:01
		io: io
	'}
	LAMP_C1_GHC_01 : FB_MKS909;

(*Normally Closed Valve with Readback*)
	{attribute 'TcLinkTo' := 	'.i_xOpnLS	:=	TIIB[LAMP_PNL2_EP25_EP2338-0002]^Channel 1^Input;
								 .i_xClsLS	:=	TIIB[LAMP_PNL2_EP25_EP2338-0002]^Channel 2^Input;
								 .q_xOPN_DO	:=	TIIB[LAMP_PNL2_EP25_EP2338-0002]^Channel 11^Output
	'}
	{attribute 'pytmc' := '
		pv: LAMP:ROUGH:VRC:01
		io: io
	'}
	LAMP_ROUGH_VRC_01 : FB_VRC;
	
	{attribute 'TcLinkTo' := 	'.i_xOpnLS	:=	TIIB[LAMP_PNL2_EP26_EP2338-0002]^Channel 1^Input;
								 .i_xClsLS	:=	TIIB[LAMP_PNL2_EP26_EP2338-0002]^Channel 2^Input;
								 .q_xOPN_DO	:=	TIIB[LAMP_PNL2_EP26_EP2338-0002]^Channel 11^Output
	'}
	{attribute 'pytmc' := '
		pv: LAMP:ROUGH:VRC:03
		io: io
	'}
	LAMP_ROUGH_VRC_03 : FB_VRC;

(*Normally Open Valve with Readback*)
	{attribute 'TcLinkTo' := 	'.i_xOpnLS	:=	TIIB[LAMP_PNL2_EP25_EP2338-0002]^Channel 5^Input;
								 .i_xClsLS	:=	TIIB[LAMP_PNL2_EP25_EP2338-0002]^Channel 6^Input;
								 .q_xCLS_DO	:=	TIIB[LAMP_PNL2_EP25_EP2338-0002]^Channel 15^Output
	'}
	{attribute 'pytmc' := '
		pv: LAMP:ROUGH:VRC:02
		io: io
	'}
	LAMP_ROUGH_VRC_02 : FB_VRC_NO;
	
(*Pfeiffer*)
	// They share the same serial port
	st_Pfeiffer_CTRL_LAMP_C2_PTM_01 		: ARRAY[1..20] OF ST_PfeifferControl;
	st_Pfeiffer_RBK_LAMP_C2_PTM_01 			: ARRAY[1..20] OF ST_PfeifferStatus;
	fb_PfeifferCom_LAMP_C2_PTM_01 			: FB_PFEIFFER_COM;
	
	st_Pfeiffer_CTRL_LAMP_C2_PTM_02 		: ARRAY[1..20] OF ST_PfeifferControl;
	st_Pfeiffer_RBK_LAMP_C2_PTM_02 			: ARRAY[1..20] OF ST_PfeifferStatus;
	fb_PfeifferCom_LAMP_C2_PTM_02 			: FB_PFEIFFER_COM;
	
	st_Pfeiffer_CTRL_LAMP_C2_PTM_03 		: ARRAY[1..20] OF ST_PfeifferControl;
	st_Pfeiffer_RBK_LAMP_C2_PTM_03 			: ARRAY[1..20] OF ST_PfeifferStatus;
	fb_PfeifferCom_LAMP_C2_PTM_03 			: FB_PFEIFFER_COM;
	
	st_Pfeiffer_CTRL_LAMP_C2_PTM_04			: ARRAY[1..20] OF ST_PfeifferControl;
	st_Pfeiffer_RBK_LAMP_C2_PTM_04 			: ARRAY[1..20] OF ST_PfeifferStatus;
	fb_PfeifferCom_LAMP_C2_PTM_04 			: FB_PFEIFFER_COM;
	
	st_Pfeiffer_CTRL_LAMP_ROUGH_PTM_01 		: ARRAY[1..20] OF ST_PfeifferControl;
	st_Pfeiffer_RBK_LAMP_ROUGH_PTM_01 		: ARRAY[1..20] OF ST_PfeifferStatus;
	fb_PfeifferCom_LAMP_ROUGH_PTM_01 		: FB_PFEIFFER_COM;
	
	st_Pfeiffer_CTRL_LAMP_C1_PTM_01 		: ARRAY[1..20] OF ST_PfeifferControl;
	st_Pfeiffer_RBK_LAMP_C1_PTM_01 			: ARRAY[1..20] OF ST_PfeifferStatus;
	fb_PfeifferCom_LAMP_C1_PTM_01 			: FB_PFEIFFER_COM;
	
	st_Pfeiffer_CTRL_LAMP_CATCH_PTM_01 		: ARRAY[1..20] OF ST_PfeifferControl;
	st_Pfeiffer_RBK_LAMP_CATCH_PTM_01 		: ARRAY[1..20] OF ST_PfeifferStatus;
	fb_PfeifferCom_LAMP_CATCH_PTM_01 		: FB_PFEIFFER_COM;
	
	st_Pfeiffer_CTRL_LAMP_CATCH_PTM_02 		: ARRAY[1..20] OF ST_PfeifferControl;
	st_Pfeiffer_RBK_LAMP_CATCH_PTM_02 		: ARRAY[1..20] OF ST_PfeifferStatus;
	fb_PfeifferCom_LAMP_CATCH_PTM_02 		: FB_PFEIFFER_COM;

	// Cluster Source - LV17 configuration
	st_Pfeiffer_CTRL_LAMP_CLSTR1_PTM_01 		: ARRAY[1..20] OF ST_PfeifferControl;
	st_Pfeiffer_RBK_LAMP_CLSTR1_PTM_01 			: ARRAY[1..20] OF ST_PfeifferStatus;
	fb_PfeifferCom_LAMP_CLSTR1_PTM_01 			: FB_PFEIFFER_COM;
	
	st_Pfeiffer_CTRL_LAMP_CLSTR1_PTM_02 		: ARRAY[1..20] OF ST_PfeifferControl;
	st_Pfeiffer_RBK_LAMP_CLSTR1_PTM_02 			: ARRAY[1..20] OF ST_PfeifferStatus;
	fb_PfeifferCom_LAMP_CLSTR1_PTM_02 			: FB_PFEIFFER_COM;
	
	st_Pfeiffer_CTRL_LAMP_CLSTR1_PTM_03 		: ARRAY[1..20] OF ST_PfeifferControl;
	st_Pfeiffer_RBK_LAMP_CLSTR1_PTM_03 			: ARRAY[1..20] OF ST_PfeifferStatus;
	fb_PfeifferCom_LAMP_CLSTR1_PTM_03 			: FB_PFEIFFER_COM;
(*	
	st_Pfeiffer_CTRL_KTOF_PTM_01 			: ARRAY[1..20] OF ST_PfeifferControl;
	st_Pfeiffer_RBK_KTOF_PTM_01 			: ARRAY[1..20] OF ST_PfeifferStatus;
	fb_PfeifferCom_KTOF_PTM_01 				: FB_PFEIFFER_COM;
*)	
	//Leybold status
	// GJ1 Turbos not connected for LV17 configuration

END_VAR

// ---- POUs/MAIN.TcPOU
PROGRAM MAIN
VAR
	
	fbLogHandler : FB_LogHandler;
	
//TMO Interface
xEcatBridge_COM_ERROR : BOOL;

(*
ITF_TMO_ROUGH1_VRC_01: FB_TVGC_2S_ADS; //FB for accessing "TMO_ROUGH1_VRC_01" VGC_2S data from PLC-TMO-VAC
ITF_TMO_ROUGH2_VRC_01: FB_TVGC_2S_ADS; //FB for accessing "TMO_ROUGH2_VRC_01" VGC_2S data from PLC-TMO-VAC
i_iWatchdog	:	UDINT; // PLC-TMO-VAC will write to this Watchdog variable
*)
b_TurboPumpRunningFlag : BOOL;
TurboPumpTOF : TOF;
TurboPumpDelayTime : TIME := T#30s;
b_PumpRunning : BOOL;
	
	ITF_TMO_ROUGH2_VRC_01: INT;
	VGC: INT;
	ITF_TMO_ROUGH1_VRC_01: INT;
	iq_stRoughRoughValve_NC_xOpnLS: INT;
	iq_stRoughRoughValve_NC_second_xOpenLS: INT;
	iq_stRoughRoughValve_NC: INT;
	iq_stRoughRoughValve_NC_second: INT;
	q_stRoughRoughValve_NC_xOpnLS: INT;
END_VAR

fbLogHandler();

// Run the Diagnostics PRG
DIAGNOSTICS();

(*
(*PLC-TMO-VAC ADS interface*)
//Writes watchdog bit to remote vac_TMO reading the vacuum components
fb_ADS_WATCHDOG_VAC_LAMP_TMO(
	sNetId:= '172.21.132.22.1.1', 
	nPort:= 851, 
	sVarName:= 'PRG_ADS_Interfaces.i_iWatchdog', 
	bError=> );
	
ITF_TMO_ROUGH1_VRC_01(//Roughing valve Readback from IP1 Roughing Line
	sNetId:= '172.21.132.22.1.1', 
	nPort:= 851, 
	sVarName:= 'GVL_Hutch_Valves.TMO_ROUGH1_VRC_01', 
	iWatchdog:= i_iWatchdog, 
	VGC=> , 
	bError=> );
	
ITF_TMO_ROUGH2_VRC_01(//Roughing valve Readback from the Gas Jet Roughing Line
	sNetId:= '172.21.132.22.1.1', 
	nPort:= 851, 
	sVarName:= 'GVL_Hutch_Valves.TMO_ROUGH2_VRC_01', 
	iWatchdog:= i_iWatchdog, 
	VGC=> , 
	bError=> );
*)

(*EtherCAT Bridge Status*)
//xEcatBridge_COM_ERROR := True means that there is an EtherCAT Bridge Communication Error.
xEcatBridge_COM_ERROR := (xEcatBridge_TxPDO_state OR xEcatBridge_External_device_not_connected OR xEcatBridge_WcState);
xOnBeamline := (xEcatBridge_COM_ERROR = FALSE) AND (sHUTCH_PLC_NAME = 'TMO');

(*TurboPump running Flag with 30 second Turn Off delay.*)
b_TurboPumpRunningFlag := (
//	(LAMP_C1_PTM_01.iq_stPtm.eState = E_PumpState.pumpRUNNING) AND //not used for x454
	(LAMP_C2_PTM_01.iq_stPtm.eState = E_PumpState.pumpRUNNING) AND // wasn't used for x471 & x454
	(LAMP_C2_PTM_02.iq_stPtm.eState = E_PumpState.pumpRUNNING) AND
	(LAMP_C2_PTM_03.iq_stPtm.eState = E_PumpState.pumpRUNNING) AND
	(LAMP_C2_PTM_04.iq_stPtm.eState = E_PumpState.pumpRUNNING) AND
	(LAMP_CATCH_PTM_01.iq_stPtm.eState = E_PumpState.pumpRUNNING) AND 
	(LAMP_CATCH_PTM_02.iq_stPtm.eState = E_PumpState.pumpRUNNING) AND
	(LAMP_ROUGH_PTM_01.iq_stPtm.eState = E_PumpState.pumpRUNNING) AND
	(LAMP_CLSTR1_PTM_01.iq_stPtm.eState = E_PumpState.pumpRUNNING) AND // Cluster Source LV17
	(LAMP_CLSTR1_PTM_02.iq_stPtm.eState = E_PumpState.pumpRUNNING) AND // Cluster Source LV17
	(LAMP_CLSTR1_PTM_03.iq_stPtm.eState = E_PumpState.pumpRUNNING));   // Cluster Source LV17
//	(KTOF_PTM_01.iq_stPtm.eState = E_PumpState.pumpRUNNING);	
TurboPumpTOF(IN:= b_TurboPumpRunningFlag, PT := TurboPumpDelayTime);
b_PumpRunning:= TurboPumpTOF.Q;
xIP1_TURBOS_ALL_AtSpd:=b_PumpRunning;

(*High Voltage Saftey Loop*)// rHighVoltageMinPressure = 1e-05; (*Hard coded High voltage Minimum Enable Pressure*)
xHighVoltageSafteyLoopEnable:= (LAMP_C2_GCC_01.IG.rPRESS <= rHighVoltageMinPressure) AND (LAMP_C2_GCC_01.IG.xPRESS_OK = TRUE);

(*PIRANI Gauges*)
	LAMP_C2_GPI_01(PG=>);
	//LAMP_CATCH_GPI_01(PG=>); which is not installed
	LAMP_GJ2_GPI_01(PG=>);
	LAMP_GJ1_GPI_01(PG=>);

(*uPIRANI Gauges*)
	LAMP_ROUGH_GPI_01(PG=>);
	LAMP_ROUGH_GPI_01.M_SetBits(32767);
	LAMP_ROUGH_GPI_02(PG=>);
	LAMP_ROUGH_GPI_02.M_SetBits(32767);
	LAMP_ROUGH_GPI_03(PG=>);
	LAMP_ROUGH_GPI_03.M_SetBits(32767);
	LAMP_ROUGH_GPI_04(PG=>);
	LAMP_ROUGH_GPI_04.M_SetBits(32767);	

(*Cold Cathode Gauges*)
	LAMP_C2_GCC_01(PG:=LAMP_C2_GPI_01.PG,IG=>,bEP:=TRUE);
	LAMP_CATCH_GCC_01(PG:=LAMP_C2_GPI_01.PG,IG=>,bEP:=TRUE);
	LAMP_CATCH_GCC_02(PG:=LAMP_C2_GPI_01.PG,IG=>,bEP:=TRUE);
	LAMP_GJ1_GCC_01(PG:=LAMP_GJ1_GPI_01.PG,IG=>,bEP:=TRUE);
	LAMP_GJ2_GCC_01(PG:=LAMP_GJ2_GPI_01.PG,IG=>,bEP:=TRUE);
	
(*Hot Cathode Gauges*)
	LAMP_C1_GHC_01(PG:=LAMP_C2_GPI_01.PG,IG=>);
	
(*TURBO Pumps
*In general, if turbo pump setpoints are above the pirani guage readings or there is no downstream open path to a roughing pump, the turbo pump will close.
*
*)
	LAMP_C1_PTM_01(
	i_xExtILKOk:= F_Turbo_NC_NO_Valve_Logic(
					i_stTurbo:= LAMP_C1_PTM_01.iq_stPtm, 
					i_stISG:= LAMP_C2_GPI_01.PG, 
					i_stBSG:= LAMP_ROUGH_GPI_02.PG, 
					iq_stValve_NO:= LAMP_ROUGH_VRC_02.iq_stValve, 
					iq_stValve_NC:= LAMP_ROUGH_VRC_01.iq_stValve, 
					iq_stValve_NC_second:= LAMP_ROUGH_VRC_03.iq_stValve,
					EcatBridge_Error_Present:= xEcatBridge_COM_ERROR,
//					ads_Error_Present:= (ITF_TMO_ROUGH1_VRC_01.bError OR ITF_TMO_ROUGH2_VRC_01.bError),
//					iq_stRoughRoughValve_NC:= ITF_TMO_ROUGH1_VRC_01.VGC,
//					iq_stRoughRoughValve_NC_second:=ITF_TMO_ROUGH2_VRC_01.VGC,
					iq_stRoughRoughValve_NC_xOpnLS:= xTMO_ROUGH1_VRC_01_OPEN_LS,
					iq_stRoughRoughValve_NC_second_xOpenLS:=xTMO_ROUGH2_VRC_01_OPEN_LS,
					x_onBeamline:= xOnBeamline), 
	iq_stPtm=> );
	
	LAMP_C2_PTM_01(
	i_xExtILKOk:= F_Turbo_NC_NO_Valve_Logic(
					i_stTurbo:= LAMP_C2_PTM_01.iq_stPtm, 
					i_stISG:= LAMP_C2_GPI_01.PG, 
					i_stBSG:= LAMP_ROUGH_GPI_02.PG, 
					iq_stValve_NO:= LAMP_ROUGH_VRC_02.iq_stValve, 
					iq_stValve_NC:= LAMP_ROUGH_VRC_01.iq_stValve, 
					iq_stValve_NC_second:= LAMP_ROUGH_VRC_03.iq_stValve,
					EcatBridge_Error_Present:= xEcatBridge_COM_ERROR,
//					ads_Error_Present:= (ITF_TMO_ROUGH1_VRC_01.bError OR ITF_TMO_ROUGH2_VRC_01.bError),
//					iq_stRoughRoughValve_NC:= ITF_TMO_ROUGH1_VRC_01.VGC,
//					iq_stRoughRoughValve_NC_second:=ITF_TMO_ROUGH2_VRC_01.VGC,
					iq_stRoughRoughValve_NC_xOpnLS:= xTMO_ROUGH1_VRC_01_OPEN_LS,
					iq_stRoughRoughValve_NC_second_xOpenLS:= xTMO_ROUGH2_VRC_01_OPEN_LS,
					x_onBeamline:= xOnBeamline), 
	iq_stPtm=> );
	
	LAMP_C2_PTM_02(
	i_xExtILKOk:= F_Turbo_NC_NO_Valve_Logic(
					i_stTurbo:= LAMP_C2_PTM_02.iq_stPtm, 
					i_stISG:= LAMP_C2_GPI_01.PG, 
					i_stBSG:= LAMP_ROUGH_GPI_02.PG, 
					iq_stValve_NO:= LAMP_ROUGH_VRC_02.iq_stValve, 
					iq_stValve_NC:= LAMP_ROUGH_VRC_01.iq_stValve, 
					iq_stValve_NC_second:= LAMP_ROUGH_VRC_03.iq_stValve,
					EcatBridge_Error_Present:= xEcatBridge_COM_ERROR,
//					ads_Error_Present:= (ITF_TMO_ROUGH1_VRC_01.bError OR ITF_TMO_ROUGH2_VRC_01.bError),
//					iq_stRoughRoughValve_NC:= ITF_TMO_ROUGH1_VRC_01.VGC,
//					iq_stRoughRoughValve_NC_second:=ITF_TMO_ROUGH2_VRC_01.VGC,
					iq_stRoughRoughValve_NC_xOpnLS:= xTMO_ROUGH1_VRC_01_OPEN_LS,
					iq_stRoughRoughValve_NC_second_xOpenLS:=xTMO_ROUGH2_VRC_01_OPEN_LS,
					x_onBeamline:= xOnBeamline), 
	iq_stPtm=> );
	
	LAMP_C2_PTM_03(
	i_xExtILKOk:= F_Turbo_NC_NO_Valve_Logic(
					i_stTurbo:= LAMP_C2_PTM_03.iq_stPtm, 
					i_stISG:= LAMP_C2_GPI_01.PG, 
					i_stBSG:= LAMP_ROUGH_GPI_02.PG, 
					iq_stValve_NO:= LAMP_ROUGH_VRC_02.iq_stValve, 
					iq_stValve_NC:= LAMP_ROUGH_VRC_01.iq_stValve, 
					iq_stValve_NC_second:= LAMP_ROUGH_VRC_03.iq_stValve,
					EcatBridge_Error_Present:= xEcatBridge_COM_ERROR,
//					ads_Error_Present:= (ITF_TMO_ROUGH1_VRC_01.bError OR ITF_TMO_ROUGH2_VRC_01.bError),
//					iq_stRoughRoughValve_NC:= ITF_TMO_ROUGH1_VRC_01.VGC,
//					iq_stRoughRoughValve_NC_second:=ITF_TMO_ROUGH2_VRC_01.VGC,
					iq_stRoughRoughValve_NC_xOpnLS:= xTMO_ROUGH1_VRC_01_OPEN_LS,
					iq_stRoughRoughValve_NC_second_xOpenLS:=xTMO_ROUGH2_VRC_01_OPEN_LS,
					x_onBeamline:= xOnBeamline), 
	iq_stPtm=> );
	
	LAMP_C2_PTM_04(
	i_xExtILKOk:= F_Turbo_NC_NO_Valve_Logic(
					i_stTurbo:= LAMP_C2_PTM_04.iq_stPtm, 
					i_stISG:= LAMP_C2_GPI_01.PG, 
					i_stBSG:= LAMP_ROUGH_GPI_02.PG, 
					iq_stValve_NO:= LAMP_ROUGH_VRC_02.iq_stValve, 
					iq_stValve_NC:= LAMP_ROUGH_VRC_01.iq_stValve, 
					iq_stValve_NC_second:= LAMP_ROUGH_VRC_03.iq_stValve,
					EcatBridge_Error_Present:= xEcatBridge_COM_ERROR,
//					ads_Error_Present:= (ITF_TMO_ROUGH1_VRC_01.bError OR ITF_TMO_ROUGH2_VRC_01.bError),
//					iq_stRoughRoughValve_NC:= ITF_TMO_ROUGH1_VRC_01.VGC,
//					iq_stRoughRoughValve_NC_second:=ITF_TMO_ROUGH2_VRC_01.VGC,
					iq_stRoughRoughValve_NC_xOpnLS:= xTMO_ROUGH1_VRC_01_OPEN_LS,
					iq_stRoughRoughValve_NC_second_xOpenLS:=xTMO_ROUGH2_VRC_01_OPEN_LS,
					x_onBeamline:= xOnBeamline), 
	iq_stPtm=> );
	
	LAMP_CATCH_PTM_01(
	i_xExtILKOk:= F_Turbo_NC_NO_Valve_Logic(
					i_stTurbo:= LAMP_CATCH_PTM_01.iq_stPtm, 
					i_stISG:= LAMP_C2_GPI_01.PG, 
					i_stBSG:= LAMP_ROUGH_GPI_02.PG, 
					iq_stValve_NO:= LAMP_ROUGH_VRC_02.iq_stValve, 
					iq_stValve_NC:= LAMP_ROUGH_VRC_01.iq_stValve, 
					iq_stValve_NC_second:= LAMP_ROUGH_VRC_03.iq_stValve,
					EcatBridge_Error_Present:= xEcatBridge_COM_ERROR,
//					ads_Error_Present:= (ITF_TMO_ROUGH1_VRC_01.bError OR ITF_TMO_ROUGH2_VRC_01.bError),
//					iq_stRoughRoughValve_NC:= ITF_TMO_ROUGH1_VRC_01.VGC,
//					iq_stRoughRoughValve_NC_second:=ITF_TMO_ROUGH2_VRC_01.VGC,
					iq_stRoughRoughValve_NC_xOpnLS:= xTMO_ROUGH1_VRC_01_OPEN_LS,
					iq_stRoughRoughValve_NC_second_xOpenLS:=xTMO_ROUGH2_VRC_01_OPEN_LS,
					x_onBeamline:= xOnBeamline), 
	iq_stPtm=> );
	
	LAMP_CATCH_PTM_02(
	i_xExtILKOk:= F_Turbo_NC_NO_Valve_Logic(
					i_stTurbo:= LAMP_CATCH_PTM_02.iq_stPtm, 
					i_stISG:= LAMP_C2_GPI_01.PG, 
					i_stBSG:= LAMP_ROUGH_GPI_02.PG, 
					iq_stValve_NO:= LAMP_ROUGH_VRC_02.iq_stValve, 
					iq_stValve_NC:= LAMP_ROUGH_VRC_01.iq_stValve, 
					iq_stValve_NC_second:= LAMP_ROUGH_VRC_03.iq_stValve,
					EcatBridge_Error_Present:= xEcatBridge_COM_ERROR,
//					ads_Error_Present:= (ITF_TMO_ROUGH1_VRC_01.bError OR ITF_TMO_ROUGH2_VRC_01.bError),
//					iq_stRoughRoughValve_NC:= ITF_TMO_ROUGH1_VRC_01.VGC,
//					iq_stRoughRoughValve_NC_second:=ITF_TMO_ROUGH2_VRC_01.VGC,
					iq_stRoughRoughValve_NC_xOpnLS:= xTMO_ROUGH1_VRC_01_OPEN_LS,
					iq_stRoughRoughValve_NC_second_xOpenLS:=xTMO_ROUGH2_VRC_01_OPEN_LS,
					x_onBeamline:= xOnBeamline), 
	iq_stPtm=> );
	
	LAMP_ROUGH_PTM_01(
	i_xExtILKOk:= F_Turbo_NC_NO_Valve_Logic(
					i_stTurbo:= LAMP_ROUGH_PTM_01.iq_stPtm, 
					i_stISG:= LAMP_C2_GPI_01.PG, 
					i_stBSG:= LAMP_ROUGH_GPI_02.PG, 
					iq_stValve_NO:= LAMP_ROUGH_VRC_02.iq_stValve, 
					iq_stValve_NC:= LAMP_ROUGH_VRC_01.iq_stValve, 
					iq_stValve_NC_second:= LAMP_ROUGH_VRC_03.iq_stValve,
					EcatBridge_Error_Present:= xEcatBridge_COM_ERROR,
//					ads_Error_Present:= (ITF_TMO_ROUGH1_VRC_01.bError OR ITF_TMO_ROUGH2_VRC_01.bError),
//					iq_stRoughRoughValve_NC:= ITF_TMO_ROUGH1_VRC_01.VGC,
//					iq_stRoughRoughValve_NC_second:=ITF_TMO_ROUGH2_VRC_01.VGC,
					iq_stRoughRoughValve_NC_xOpnLS:= xTMO_ROUGH1_VRC_01_OPEN_LS,
					iq_stRoughRoughValve_NC_second_xOpenLS:=xTMO_ROUGH2_VRC_01_OPEN_LS,
					x_onBeamline:= xOnBeamline), 
	iq_stPtm=> );

// Cluster Source - LV17 Configuration
	LAMP_CLSTR1_PTM_01(
	i_xExtILKOk:= F_Turbo_NC_NO_Valve_Logic(
					i_stTurbo:= LAMP_CLSTR1_PTM_01.iq_stPtm, 
					i_stISG:= LAMP_GJ1_GPI_01.PG, 
					i_stBSG:= LAMP_ROUGH_GPI_04.PG, 
					iq_stValve_NO:= LAMP_ROUGH_VRC_02.iq_stValve, 
					iq_stValve_NC:= LAMP_ROUGH_VRC_03.iq_stValve, 
					iq_stValve_NC_second:= LAMP_ROUGH_VRC_01.iq_stValve,
					EcatBridge_Error_Present:= xEcatBridge_COM_ERROR,
					iq_stRoughRoughValve_NC_xOpnLS:= xTMO_ROUGH2_VRC_01_OPEN_LS,
					iq_stRoughRoughValve_NC_second_xOpenLS:=xTMO_ROUGH1_VRC_01_OPEN_LS,
					x_onBeamline:= xOnBeamline), 
	iq_stPtm=> );
	
	LAMP_CLSTR1_PTM_02(
	i_xExtILKOk:= F_Turbo_NC_NO_Valve_Logic(
					i_stTurbo:= LAMP_CLSTR1_PTM_02.iq_stPtm, 
					i_stISG:= LAMP_GJ1_GPI_01.PG, 
					i_stBSG:= LAMP_ROUGH_GPI_04.PG, 
					iq_stValve_NO:= LAMP_ROUGH_VRC_02.iq_stValve, 
					iq_stValve_NC:= LAMP_ROUGH_VRC_03.iq_stValve, 
					iq_stValve_NC_second:= LAMP_ROUGH_VRC_01.iq_stValve,
					EcatBridge_Error_Present:= xEcatBridge_COM_ERROR,
					iq_stRoughRoughValve_NC_xOpnLS:= xTMO_ROUGH2_VRC_01_OPEN_LS,
					iq_stRoughRoughValve_NC_second_xOpenLS:=xTMO_ROUGH1_VRC_01_OPEN_LS,
					x_onBeamline:= xOnBeamline), 
	iq_stPtm=> );
	
	LAMP_CLSTR1_PTM_03(
	i_xExtILKOk:= F_Turbo_NC_NO_Valve_Logic(
					i_stTurbo:= LAMP_CLSTR1_PTM_03.iq_stPtm, 
					i_stISG:= LAMP_GJ1_GPI_01.PG, 
					i_stBSG:= LAMP_ROUGH_GPI_04.PG, 
					iq_stValve_NO:= LAMP_ROUGH_VRC_02.iq_stValve, 
					iq_stValve_NC:= LAMP_ROUGH_VRC_03.iq_stValve, 
					iq_stValve_NC_second:= LAMP_ROUGH_VRC_01.iq_stValve,
					EcatBridge_Error_Present:= xEcatBridge_COM_ERROR,
					iq_stRoughRoughValve_NC_xOpnLS:= xTMO_ROUGH1_VRC_01_OPEN_LS,
					iq_stRoughRoughValve_NC_second_xOpenLS:=xTMO_ROUGH2_VRC_01_OPEN_LS,
					x_onBeamline:= xOnBeamline), 
	iq_stPtm=> );
	
(*	
	KTOF_PTM_01(
	i_xExtILKOk:= F_Turbo_NC_NO_Valve_Logic(
					i_stTurbo:= KTOF_PTM_01.iq_stPtm, 
					i_stISG:= LAMP_C2_GPI_01.PG, 
					i_stBSG:= LAMP_ROUGH_GPI_02.PG, 
					iq_stValve_NO:= LAMP_ROUGH_VRC_02.iq_stValve, 
					iq_stValve_NC:= LAMP_ROUGH_VRC_01.iq_stValve, 
					iq_stValve_NC_second:= LAMP_ROUGH_VRC_03.iq_stValve,
					EcatBridge_Error_Present:= xEcatBridge_COM_ERROR,
//					ads_Error_Present:= (ITF_TMO_ROUGH1_VRC_01.bError OR ITF_TMO_ROUGH2_VRC_01.bError),
					iq_stRoughRoughValve_NC:= ITF_TMO_ROUGH1_VRC_01.VGC,
					iq_stRoughRoughValve_NC_second:=ITF_TMO_ROUGH2_VRC_01.VGC,
					x_onBeamline:= xOnBeamline), 
	iq_stPtm=> );
*)	
(*Serial Communication*)
(*Assign adresses to the pfeiffer controllers connected to this serial terminal*)
//LAMP:C2:PTM:01
st_Pfeiffer_CTRL_LAMP_C2_PTM_01[1].iSerialAddress :=1;
st_Pfeiffer_CTRL_LAMP_C2_PTM_01[1].xEnableComm := TRUE;
(* Instanitate the Function block for serial communication with Pfeiffer*)	
fb_PfeifferCom_LAMP_C2_PTM_01(astPfeifferControl := st_Pfeiffer_CTRL_LAMP_C2_PTM_01,
			   				  astPfeifferStatus:= st_Pfeiffer_RBK_LAMP_C2_PTM_01,
							  SerialRXBuffer:= SerialRXBuffer_LAMP_C2_PTM_01,
							  SerialTXBuffer:= SerialTXBuffer_LAMP_C2_PTM_01);
(* Copy Status Pv's into the PTM structure*)
LAMP_C2_PTM_01.M_Serial_IO(st_Pfeiffer_RBK:= st_Pfeiffer_RBK_LAMP_C2_PTM_01[1], st_Pfeiffer_CTRL:= st_Pfeiffer_CTRL_LAMP_C2_PTM_01[1]);

//LAMP:C2:PTM:02
st_Pfeiffer_CTRL_LAMP_C2_PTM_02[1].iSerialAddress :=1;
st_Pfeiffer_CTRL_LAMP_C2_PTM_02[1].xEnableComm := TRUE;
fb_PfeifferCom_LAMP_C2_PTM_02(astPfeifferControl := st_Pfeiffer_CTRL_LAMP_C2_PTM_02,
			   				  astPfeifferStatus:= st_Pfeiffer_RBK_LAMP_C2_PTM_02,
							  SerialRXBuffer:= SerialRXBuffer_LAMP_C2_PTM_02,
							  SerialTXBuffer:= SerialTXBuffer_LAMP_C2_PTM_02);
LAMP_C2_PTM_02.M_Serial_IO(st_Pfeiffer_RBK:= st_Pfeiffer_RBK_LAMP_C2_PTM_02[1], st_Pfeiffer_CTRL:= st_Pfeiffer_CTRL_LAMP_C2_PTM_02[1]);

//LAMP:C2:PTM:03
st_Pfeiffer_CTRL_LAMP_C2_PTM_03[1].iSerialAddress :=1;
st_Pfeiffer_CTRL_LAMP_C2_PTM_03[1].xEnableComm := TRUE;
fb_PfeifferCom_LAMP_C2_PTM_03(astPfeifferControl := st_Pfeiffer_CTRL_LAMP_C2_PTM_03,
			   				  astPfeifferStatus:= st_Pfeiffer_RBK_LAMP_C2_PTM_03,
							  SerialRXBuffer:= SerialRXBuffer_LAMP_C2_PTM_03,
							  SerialTXBuffer:= SerialTXBuffer_LAMP_C2_PTM_03);
LAMP_C2_PTM_03.M_Serial_IO(st_Pfeiffer_RBK:= st_Pfeiffer_RBK_LAMP_C2_PTM_03[1], st_Pfeiffer_CTRL:= st_Pfeiffer_CTRL_LAMP_C2_PTM_03[1]);

//LAMP:C2:PTM:04
st_Pfeiffer_CTRL_LAMP_C2_PTM_04[1].iSerialAddress :=1;
st_Pfeiffer_CTRL_LAMP_C2_PTM_04[1].xEnableComm := TRUE;
fb_PfeifferCom_LAMP_C2_PTM_04(astPfeifferControl := st_Pfeiffer_CTRL_LAMP_C2_PTM_04,
			   				  astPfeifferStatus:= st_Pfeiffer_RBK_LAMP_C2_PTM_04,
							  SerialRXBuffer:= SerialRXBuffer_LAMP_C2_PTM_04,
							  SerialTXBuffer:= SerialTXBuffer_LAMP_C2_PTM_04);
LAMP_C2_PTM_04.M_Serial_IO(st_Pfeiffer_RBK:= st_Pfeiffer_RBK_LAMP_C2_PTM_04[1], st_Pfeiffer_CTRL:= st_Pfeiffer_CTRL_LAMP_C2_PTM_04[1]);

//LAMP:ROUGH:PTM:01
st_Pfeiffer_CTRL_LAMP_ROUGH_PTM_01[1].iSerialAddress :=1;
st_Pfeiffer_CTRL_LAMP_ROUGH_PTM_01[1].xEnableComm := TRUE;
fb_PfeifferCom_LAMP_ROUGH_PTM_01(astPfeifferControl := st_Pfeiffer_CTRL_LAMP_ROUGH_PTM_01,
			   				  astPfeifferStatus:= st_Pfeiffer_RBK_LAMP_ROUGH_PTM_01,
							  SerialRXBuffer:= SerialRXBuffer_LAMP_ROUGH_PTM_01,
							  SerialTXBuffer:= SerialTXBuffer_LAMP_ROUGH_PTM_01);
LAMP_ROUGH_PTM_01.M_Serial_IO(st_Pfeiffer_RBK:= st_Pfeiffer_RBK_LAMP_ROUGH_PTM_01[1], st_Pfeiffer_CTRL:= st_Pfeiffer_CTRL_LAMP_ROUGH_PTM_01[1]);

//LAMP:C1:PTM:01
st_Pfeiffer_CTRL_LAMP_C1_PTM_01[1].iSerialAddress :=1;
st_Pfeiffer_CTRL_LAMP_C1_PTM_01[1].xEnableComm := TRUE;
fb_PfeifferCom_LAMP_C1_PTM_01(astPfeifferControl := st_Pfeiffer_CTRL_LAMP_C1_PTM_01,
			   				  astPfeifferStatus:= st_Pfeiffer_RBK_LAMP_C1_PTM_01,
							  SerialRXBuffer:= SerialRXBuffer_LAMP_C1_PTM_01,
							  SerialTXBuffer:= SerialTXBuffer_LAMP_C1_PTM_01);
LAMP_C1_PTM_01.M_Serial_IO(st_Pfeiffer_RBK:= st_Pfeiffer_RBK_LAMP_C1_PTM_01[1], st_Pfeiffer_CTRL:= st_Pfeiffer_CTRL_LAMP_C1_PTM_01[1]);

//LAMP:CATCH:PTM:01
st_Pfeiffer_CTRL_LAMP_CATCH_PTM_01[1].iSerialAddress :=1;
st_Pfeiffer_CTRL_LAMP_CATCH_PTM_01[1].xEnableComm := TRUE;
fb_PfeifferCom_LAMP_CATCH_PTM_01(astPfeifferControl := st_Pfeiffer_CTRL_LAMP_CATCH_PTM_01,
			   				  astPfeifferStatus:= st_Pfeiffer_RBK_LAMP_CATCH_PTM_01,
							  SerialRXBuffer:= SerialRXBuffer_LAMP_CATCH_PTM_01,
							  SerialTXBuffer:= SerialTXBuffer_LAMP_CATCH_PTM_01);
LAMP_CATCH_PTM_01.M_Serial_IO(st_Pfeiffer_RBK:= st_Pfeiffer_RBK_LAMP_CATCH_PTM_01[1], st_Pfeiffer_CTRL:= st_Pfeiffer_CTRL_LAMP_CATCH_PTM_01[1]);

//LAMP:CATCH:PTM:02
st_Pfeiffer_CTRL_LAMP_CATCH_PTM_02[1].iSerialAddress :=1;
st_Pfeiffer_CTRL_LAMP_CATCH_PTM_02[1].xEnableComm := TRUE;
fb_PfeifferCom_LAMP_CATCH_PTM_02(astPfeifferControl := st_Pfeiffer_CTRL_LAMP_CATCH_PTM_02,
			   				  astPfeifferStatus:= st_Pfeiffer_RBK_LAMP_CATCH_PTM_02,
							  SerialRXBuffer:= SerialRXBuffer_LAMP_CATCH_PTM_02,
							  SerialTXBuffer:= SerialTXBuffer_LAMP_CATCH_PTM_02);
LAMP_CATCH_PTM_02.M_Serial_IO(st_Pfeiffer_RBK:= st_Pfeiffer_RBK_LAMP_CATCH_PTM_02[1], st_Pfeiffer_CTRL:= st_Pfeiffer_CTRL_LAMP_CATCH_PTM_02[1]);

// LAMP LV17 Cluster Source Configuration
//CLSTR1:PTM:01
st_Pfeiffer_CTRL_LAMP_CLSTR1_PTM_01[1].iSerialAddress :=1;
st_Pfeiffer_CTRL_LAMP_CLSTR1_PTM_01[1].xEnableComm := TRUE;
fb_PfeifferCom_LAMP_CLSTR1_PTM_01(astPfeifferControl := st_Pfeiffer_CTRL_LAMP_CLSTR1_PTM_01,
			   				  astPfeifferStatus:= st_Pfeiffer_RBK_LAMP_CLSTR1_PTM_01,
							  SerialRXBuffer:= SerialRXBuffer_LAMP_CLSTR1_PTM_01,
							  SerialTXBuffer:= SerialTXBuffer_LAMP_CLSTR1_PTM_01);
LAMP_CLSTR1_PTM_01.M_Serial_IO(st_Pfeiffer_RBK:= st_Pfeiffer_RBK_LAMP_CLSTR1_PTM_01[1], st_Pfeiffer_CTRL:= st_Pfeiffer_CTRL_LAMP_CLSTR1_PTM_01[1]);

//CLSTR1:PTM:02
st_Pfeiffer_CTRL_LAMP_CLSTR1_PTM_02[1].iSerialAddress :=1;
st_Pfeiffer_CTRL_LAMP_CLSTR1_PTM_02[1].xEnableComm := TRUE;
fb_PfeifferCom_LAMP_CLSTR1_PTM_02(astPfeifferControl := st_Pfeiffer_CTRL_LAMP_CLSTR1_PTM_02,
			   				  astPfeifferStatus:= st_Pfeiffer_RBK_LAMP_CLSTR1_PTM_02,
							  SerialRXBuffer:= SerialRXBuffer_LAMP_CLSTR1_PTM_02,
							  SerialTXBuffer:= SerialTXBuffer_LAMP_CLSTR1_PTM_02);
LAMP_CLSTR1_PTM_02.M_Serial_IO(st_Pfeiffer_RBK:= st_Pfeiffer_RBK_LAMP_CLSTR1_PTM_02[1], st_Pfeiffer_CTRL:= st_Pfeiffer_CTRL_LAMP_CLSTR1_PTM_02[1]);

//CLSTR1:PTM:03
st_Pfeiffer_CTRL_LAMP_CLSTR1_PTM_03[1].iSerialAddress :=1;
st_Pfeiffer_CTRL_LAMP_CLSTR1_PTM_03[1].xEnableComm := TRUE;
fb_PfeifferCom_LAMP_CLSTR1_PTM_03(astPfeifferControl := st_Pfeiffer_CTRL_LAMP_CLSTR1_PTM_03,
			   				  astPfeifferStatus:= st_Pfeiffer_RBK_LAMP_CLSTR1_PTM_03,
							  SerialRXBuffer:= SerialRXBuffer_LAMP_CLSTR1_PTM_03,
							  SerialTXBuffer:= SerialTXBuffer_LAMP_CLSTR1_PTM_03);
LAMP_CLSTR1_PTM_03.M_Serial_IO(st_Pfeiffer_RBK:= st_Pfeiffer_RBK_LAMP_CLSTR1_PTM_03[1], st_Pfeiffer_CTRL:= st_Pfeiffer_CTRL_LAMP_CLSTR1_PTM_03[1]);

(*
st_Pfeiffer_CTRL_KTOF_PTM_01[1].iSerialAddress :=1;
st_Pfeiffer_CTRL_KTOF_PTM_01[1].xEnableComm := TRUE;
fb_PfeifferCom_KTOF_PTM_01(astPfeifferControl := st_Pfeiffer_CTRL_KTOF_PTM_01,
			   				  astPfeifferStatus:= st_Pfeiffer_RBK_KTOF_PTM_01,
							  SerialRXBuffer:= SerialRXBuffer_KTOF_PTM_01,
							  SerialTXBuffer:= SerialTXBuffer_KTOF_PTM_01);
//KTOF_PTM_01.M_Serial_IO(st_Pfeiffer_CTRL_KTOF_PTM_01[1],st_Pfeiffer_RBK_KTOF_PTM_01[1]);
KTOF_PTM_01.M_Serial_IO(st_Pfeiffer_RBK:= st_Pfeiffer_RBK_KTOF_PTM_01[1], st_Pfeiffer_CTRL:= st_Pfeiffer_CTRL_KTOF_PTM_01[1]);
*)

//Leybolds
//GJ1 not included in LV17 configuration

(*Vacuum Gate Valve*)

(* Old LAMP logic
	LAMP_ROUGH_VRC_01(//LAMP:ROUGH:VRC:01 can open when the pressure across the valve is below 10 torr
	i_xExtILK_OK:= (ABS(LAMP_ROUGH_GPI_01.PG.rPRESS - LAMP_ROUGH_GPI_02.PG.rPRESS)<10.0),
	i_xOverrideMode:= xSystemOverrideMode_LAMP, 
	iq_stValve=> );
	
	LAMP_ROUGH_VRC_02(//LAMP:ROUGH:VRC:02 close when the pressure in the the C2, GJ1, and GJ2 chambers are all below 10 torr.
	i_xExtILK_OK:= NOT((LAMP_GJ1_GPI_01.PG.rPRESS >10.0) OR (LAMP_GJ2_GPI_01.PG.rPRESS > 10.0) OR (LAMP_C2_GPI_01.PG.rPRESS > 10.0)) , 
	i_xOverrideMode:= xSystemOverrideMode_LAMP, 
	iq_stValve=> );
	
	LAMP_ROUGH_VRC_03(//LAMP:ROUGH:VRC:03 can open when the pressure across the valve is below 10 torr
	i_xExtILK_OK:= (ABS(LAMP_ROUGH_GPI_03.PG.rPRESS - LAMP_ROUGH_GPI_04.PG.rPRESS)<10.0),
	i_xOverrideMode:= xSystemOverrideMode_LAMP, 
	iq_stValve=> );
*)	

(*Vacuum Gate Valve*) //LAMP MBES code 
	IF(xOnBeamline) THEN //If OnBeamline then stay open.
		LAMP_ROUGH_VRC_01.M_Set_OPN_SW(TRUE);
		LAMP_ROUGH_VRC_01(
		i_xExtILK_OK:= TRUE,
		i_xOverrideMode:= xSystemOverrideMode_LAMP,
		iq_stValve=> );
	ELSE
		LAMP_ROUGH_VRC_01(//LAMP:ROUGH:VRC:01 can open when the pressure across the valve is below 10 torr
		i_xExtILK_OK:= (ABS(LAMP_ROUGH_GPI_01.PG.rPRESS - LAMP_ROUGH_GPI_02.PG.rPRESS)<10.0),   
		i_xOverrideMode:= xSystemOverrideMode_LAMP, 
		iq_stValve=> );
	END_IF

    LAMP_ROUGH_VRC_02(//LAMP:ROUGH:VRC:02 close when the pressure in the C2, GJ1, GJ2 chambers are all below 10 torr.)
	i_xExtILK_OK:= NOT ((LAMP_ROUGH_GPI_01.PG.rPRESS > 10.0 ) OR (LAMP_ROUGH_GPI_02.PG.rPRESS > 10.0) OR (LAMP_C2_GPI_01.PG.rPRESS > 10) ), 
	i_xOverrideMode:= xSystemOverrideMode_LAMP,
 	iq_stValve=> );
	IF(xOnBeamline) THEN //If OnBeamline then stay open.
		LAMP_ROUGH_VRC_03.M_Set_OPN_SW(TRUE);
		LAMP_ROUGH_VRC_03(
		i_xExtILK_OK:= TRUE,
		i_xOverrideMode:= xSystemOverrideMode_LAMP,
		iq_stValve=> );
    ELSE
		LAMP_ROUGH_VRC_03(//LAMP:ROUGH:VRC:03 can open when the pressure across the valve is below 10 torr
		i_xExtILK_OK:= (ABS(LAMP_ROUGH_GPI_03.PG.rPRESS - LAMP_ROUGH_GPI_04.PG.rPRESS)<10.0), 
		i_xOverrideMode:= xSystemOverrideMode_LAMP, 
		iq_stValve=> );
	END_IF	


(*Update EtherCAT Bridge Outputs*)
xIP1_ROUGH_VRC_01_OPEN_LS := LAMP_ROUGH_VRC_01.M_IsOpen();
xIP1_ROUGH_VRC_02_OPEN_LS := LAMP_ROUGH_VRC_02.M_IsOpen();
xIP1_ROUGH_VRC_03_OPEN_LS := LAMP_ROUGH_VRC_03.M_IsOpen();
//xIP1_TURBO_FAULT AT %Q* : BOOL; already updated at turbo logic
xIP1_MAIN_xAT_VAC         := LAMP_C2_GCC_01.IG.xAT_VAC;
xIP1_MAIN_xPRESS_OK       := LAMP_C2_GCC_01.IG.xPRESS_OK;
rIP1_MAIN_rPRESS          := LAMP_C2_GCC_01.IG.rPRESS;
xIP1_HV_SAFETY_ENABLE     := xHighVoltageSafteyLoopEnable;

END_PROGRAM

// ---- POUs/PRG_COM.TcPOU
PROGRAM PRG_COM
VAR
END_VAR

(*Instanitate Serial port com function *) 
fbSerialLineControl_LAMP_C2_PTM_01(
	Mode:= SERIALLINEMODE_EL6_22B,
	pComIn:= ADR(stComIn_LAMP_C2_PTM_01),
	pComOut:=ADR(stComOut_LAMP_C2_PTM_01),
	SizeComIn:= SIZEOF(stComIn_LAMP_C2_PTM_01),
	TxBuffer:= SerialTXBuffer_LAMP_C2_PTM_01,
	RxBuffer:= SerialRXBuffer_LAMP_C2_PTM_01,
	Error=> ,
	ErrorID=> );
	
fbSerialLineControl_LAMP_C2_PTM_02(
	Mode:= SERIALLINEMODE_EL6_22B,
	pComIn:= ADR(stComIn_LAMP_C2_PTM_02),
	pComOut:=ADR(stComOut_LAMP_C2_PTM_02),
	SizeComIn:= SIZEOF(stComIn_LAMP_C2_PTM_02),
	TxBuffer:= SerialTXBuffer_LAMP_C2_PTM_02,
	RxBuffer:= SerialRXBuffer_LAMP_C2_PTM_02,
	Error=> ,
	ErrorID=> );
	
fbSerialLineControl_LAMP_C2_PTM_03(
	Mode:= SERIALLINEMODE_EL6_22B,
	pComIn:= ADR(stComIn_LAMP_C2_PTM_03),
	pComOut:=ADR(stComOut_LAMP_C2_PTM_03),
	SizeComIn:= SIZEOF(stComIn_LAMP_C2_PTM_03),
	TxBuffer:= SerialTXBuffer_LAMP_C2_PTM_03,
	RxBuffer:= SerialRXBuffer_LAMP_C2_PTM_03,
	Error=> ,
	ErrorID=> );
	
fbSerialLineControl_LAMP_C2_PTM_04(
	Mode:= SERIALLINEMODE_EL6_22B,
	pComIn:= ADR(stComIn_LAMP_C2_PTM_04),
	pComOut:=ADR(stComOut_LAMP_C2_PTM_04),
	SizeComIn:= SIZEOF(stComIn_LAMP_C2_PTM_04),
	TxBuffer:= SerialTXBuffer_LAMP_C2_PTM_04,
	RxBuffer:= SerialRXBuffer_LAMP_C2_PTM_04,
	Error=> ,
	ErrorID=> );
	
fbSerialLineControl_LAMP_ROUGH_PTM_01(
	Mode:= SERIALLINEMODE_EL6_22B,
	pComIn:= ADR(stComIn_LAMP_ROUGH_PTM_01),
	pComOut:=ADR(stComOut_LAMP_ROUGH_PTM_01),
	SizeComIn:= SIZEOF(stComIn_LAMP_ROUGH_PTM_01),
	TxBuffer:= SerialTXBuffer_LAMP_ROUGH_PTM_01,
	RxBuffer:= SerialRXBuffer_LAMP_ROUGH_PTM_01,
	Error=> ,
	ErrorID=> );
	
fbSerialLineControl_LAMP_C1_PTM_01(
	Mode:= SERIALLINEMODE_EL6_22B,
	pComIn:= ADR(stComIn_LAMP_C1_PTM_01),
	pComOut:=ADR(stComOut_LAMP_C1_PTM_01),
	SizeComIn:= SIZEOF(stComIn_LAMP_C1_PTM_01),
	TxBuffer:= SerialTXBuffer_LAMP_C1_PTM_01,
	RxBuffer:= SerialRXBuffer_LAMP_C1_PTM_01,
	Error=> ,
	ErrorID=> );
	
fbSerialLineControl_LAMP_CATCH_PTM_01(
	Mode:= SERIALLINEMODE_EL6_22B,
	pComIn:= ADR(stComIn_LAMP_CATCH_PTM_01),
	pComOut:=ADR(stComOut_LAMP_CATCH_PTM_01),
	SizeComIn:= SIZEOF(stComIn_LAMP_CATCH_PTM_01),
	TxBuffer:= SerialTXBuffer_LAMP_CATCH_PTM_01,
	RxBuffer:= SerialRXBuffer_LAMP_CATCH_PTM_01,
	Error=> ,
	ErrorID=> );
	
fbSerialLineControl_LAMP_CATCH_PTM_02(
	Mode:= SERIALLINEMODE_EL6_22B,
	pComIn:= ADR(stComIn_LAMP_CATCH_PTM_02),
	pComOut:=ADR(stComOut_LAMP_CATCH_PTM_02),
	SizeComIn:= SIZEOF(stComIn_LAMP_CATCH_PTM_02),
	TxBuffer:= SerialTXBuffer_LAMP_CATCH_PTM_02,
	RxBuffer:= SerialRXBuffer_LAMP_CATCH_PTM_02,
	Error=> ,
	ErrorID=> );
	
// Cluster Source - LV17 Configuration
fbSerialLineControl_LAMP_CLSTR1_PTM_01(
	Mode:= SERIALLINEMODE_EL6_22B,
	pComIn:= ADR(stComIn_LAMP_CLSTR1_PTM_01),
	pComOut:=ADR(stComOut_LAMP_CLSTR1_PTM_01),
	SizeComIn:= SIZEOF(stComIn_LAMP_CLSTR1_PTM_01),
	TxBuffer:= SerialTXBuffer_LAMP_CLSTR1_PTM_01,
	RxBuffer:= SerialRXBuffer_LAMP_CLSTR1_PTM_01,
	Error=> ,
	ErrorID=> );

fbSerialLineControl_LAMP_CLSTR1_PTM_02(
	Mode:= SERIALLINEMODE_EL6_22B,
	pComIn:= ADR(stComIn_LAMP_CLSTR1_PTM_02),
	pComOut:=ADR(stComOut_LAMP_CLSTR1_PTM_02),
	SizeComIn:= SIZEOF(stComIn_LAMP_CLSTR1_PTM_02),
	TxBuffer:= SerialTXBuffer_LAMP_CLSTR1_PTM_02,
	RxBuffer:= SerialRXBuffer_LAMP_CLSTR1_PTM_02,
	Error=> ,
	ErrorID=> );

fbSerialLineControl_LAMP_CLSTR1_PTM_03(
	Mode:= SERIALLINEMODE_EL6_22B,
	pComIn:= ADR(stComIn_LAMP_CLSTR1_PTM_03),
	pComOut:=ADR(stComOut_LAMP_CLSTR1_PTM_03),
	SizeComIn:= SIZEOF(stComIn_LAMP_CLSTR1_PTM_03),
	TxBuffer:= SerialTXBuffer_LAMP_CLSTR1_PTM_03,
	RxBuffer:= SerialRXBuffer_LAMP_CLSTR1_PTM_03,
	Error=> ,
	ErrorID=> );	
(*	
fbSerialLineControl_KTOF_PTM_01(
	Mode:= SERIALLINEMODE_EL6_22B,
	pComIn:= ADR(stComIn_KTOF_PTM_01),
	pComOut:=ADR(stComOut_KTOF_PTM_01),
	SizeComIn:= SIZEOF(stComIn_KTOF_PTM_01),
	TxBuffer:= SerialTXBuffer_KTOF_PTM_01,
	RxBuffer:= SerialRXBuffer_KTOF_PTM_01,
	Error=> ,
	ErrorID=> );
*)

END_PROGRAM
